REGION Network 79: K
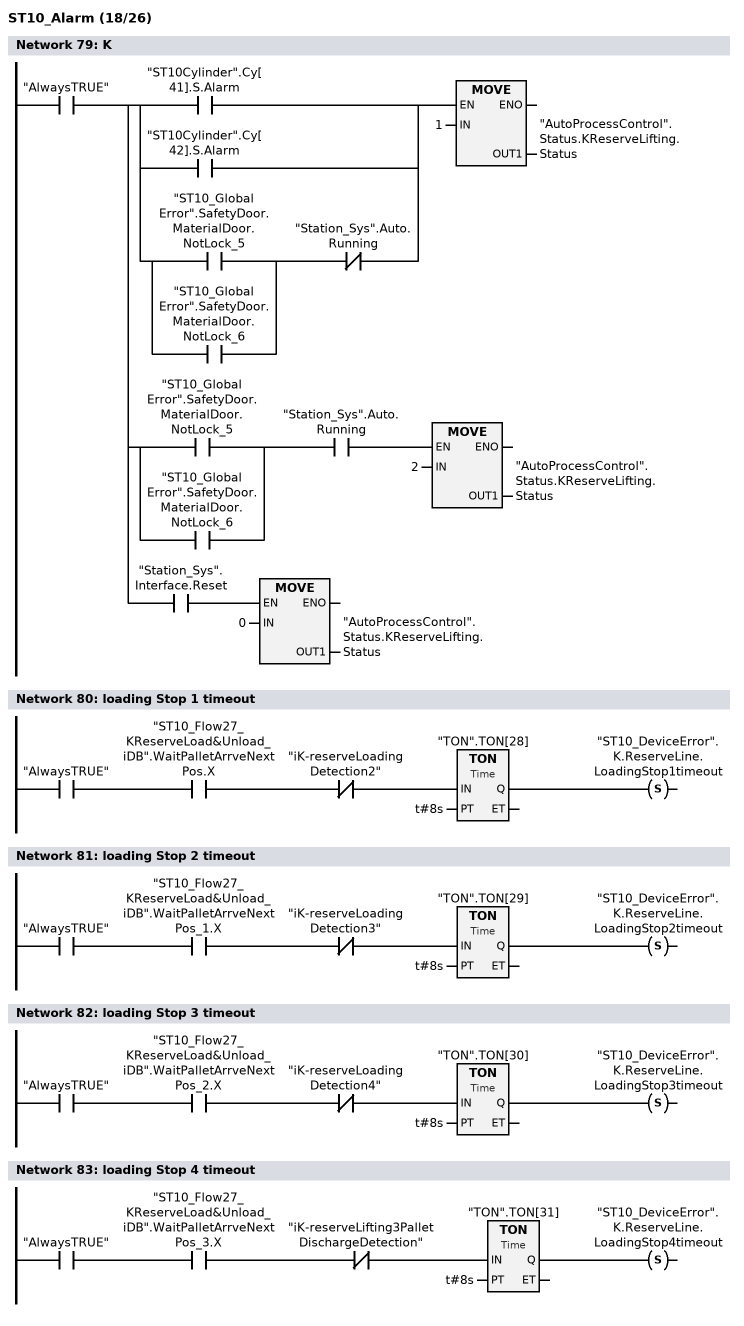
   RUNG wire#powerrail
      Contact( "AlwaysTRUE" )
      wire#w1
      Contact( "ST10Cylinder".Cy[41].S.Alarm )
      wire#w2
      Move(in := 1, out1 => "AutoProcessControl".Status.KReserveLifting.Status)
   END_RUNG
   RUNG wire#w1
      Contact( "ST10Cylinder".Cy[42].S.Alarm )
   END_RUNG wire#w2
   RUNG wire#w1
      Contact( "ST10_GlobalError".SafetyDoor.MaterialDoor.NotLock_5 )
      wire#w3
      I_Contact( "Station_Sys".Auto.Running )
   END_RUNG wire#w2
   RUNG wire#w1
      Contact( "ST10_GlobalError".SafetyDoor.MaterialDoor.NotLock_6 )
   END_RUNG wire#w3
   RUNG wire#w1
      Contact( "ST10_GlobalError".SafetyDoor.MaterialDoor.NotLock_5 )
      wire#w4
      Contact( "Station_Sys".Auto.Running )
      Move(in := 2, out1 => "AutoProcessControl".Status.KReserveLifting.Status)
   END_RUNG
   RUNG wire#w1
      Contact( "ST10_GlobalError".SafetyDoor.MaterialDoor.NotLock_6 )
   END_RUNG wire#w4
   RUNG wire#w1
      Contact( "Station_Sys".Interface.Reset )
      Move(in := 0, out1 => "AutoProcessControl".Status.KReserveLifting.Status)
   END_RUNG
   // the same network as SCL:
   IF "AlwaysTRUE" AND ("ST10Cylinder".Cy[41].S.Alarm OR "ST10Cylinder".Cy[42].S.Alarm OR (("ST10_GlobalError".SafetyDoor.MaterialDoor.NotLock_5 OR "ST10_GlobalError".SafetyDoor.MaterialDoor.NotLock_6) AND NOT "Station_Sys".Auto.Running)) THEN
       "AutoProcessControl".Status.KReserveLifting.Status := 1;
   END_IF;
   IF "AlwaysTRUE" AND ("ST10_GlobalError".SafetyDoor.MaterialDoor.NotLock_5 OR "ST10_GlobalError".SafetyDoor.MaterialDoor.NotLock_6) AND "Station_Sys".Auto.Running THEN
       "AutoProcessControl".Status.KReserveLifting.Status := 2;
   END_IF;
   IF "AlwaysTRUE" AND "Station_Sys".Interface.Reset THEN
       "AutoProcessControl".Status.KReserveLifting.Status := 0;
   END_IF;
END_REGION

REGION Network 80: loading Stop 1 timeout
   RUNG wire#powerrail
      Contact( "AlwaysTRUE" )
      Contact( "ST10_Flow27_KReserveLoad&Unload_iDB".WaitPalletArrveNextPos.X )
      I_Contact( "iK-reserveLoadingDetection2" )
      { S7_Templates := "time_type := Time" } "TON".TON[28].TON(pt := t#8s, et =>)
      S_Coil( "ST10_DeviceError".K.ReserveLine.LoadingStop1timeout )
   END_RUNG
   // the same network as SCL:
   "TON".TON[28].TON(IN := "AlwaysTRUE" AND "ST10_Flow27_KReserveLoad&Unload_iDB".WaitPalletArrveNextPos.X AND NOT "iK-reserveLoadingDetection2",
                     PT := t#8s);
   IF "TON".TON[28].Q THEN "ST10_DeviceError".K.ReserveLine.LoadingStop1timeout := TRUE; END_IF;
END_REGION

REGION Network 81: loading Stop 2 timeout
   RUNG wire#powerrail
      Contact( "AlwaysTRUE" )
      Contact( "ST10_Flow27_KReserveLoad&Unload_iDB".WaitPalletArrveNextPos_1.X )
      I_Contact( "iK-reserveLoadingDetection3" )
      { S7_Templates := "time_type := Time" } "TON".TON[29].TON(pt := t#8s, et =>)
      S_Coil( "ST10_DeviceError".K.ReserveLine.LoadingStop2timeout )
   END_RUNG
   // the same network as SCL:
   "TON".TON[29].TON(IN := "AlwaysTRUE" AND "ST10_Flow27_KReserveLoad&Unload_iDB".WaitPalletArrveNextPos_1.X AND NOT "iK-reserveLoadingDetection3",
                     PT := t#8s);
   IF "TON".TON[29].Q THEN "ST10_DeviceError".K.ReserveLine.LoadingStop2timeout := TRUE; END_IF;
END_REGION

REGION Network 82: loading Stop 3 timeout
   RUNG wire#powerrail
      Contact( "AlwaysTRUE" )
      Contact( "ST10_Flow27_KReserveLoad&Unload_iDB".WaitPalletArrveNextPos_2.X )
      I_Contact( "iK-reserveLoadingDetection4" )
      { S7_Templates := "time_type := Time" } "TON".TON[30].TON(pt := t#8s, et =>)
      S_Coil( "ST10_DeviceError".K.ReserveLine.LoadingStop3timeout )
   END_RUNG
   // the same network as SCL:
   "TON".TON[30].TON(IN := "AlwaysTRUE" AND "ST10_Flow27_KReserveLoad&Unload_iDB".WaitPalletArrveNextPos_2.X AND NOT "iK-reserveLoadingDetection4",
                     PT := t#8s);
   IF "TON".TON[30].Q THEN "ST10_DeviceError".K.ReserveLine.LoadingStop3timeout := TRUE; END_IF;
END_REGION

REGION Network 83: loading Stop 4 timeout
   RUNG wire#powerrail
      Contact( "AlwaysTRUE" )
      Contact( "ST10_Flow27_KReserveLoad&Unload_iDB".WaitPalletArrveNextPos_3.X )
      I_Contact( "iK-reserveLifting3PalletDischargeDetection" )
      { S7_Templates := "time_type := Time" } "TON".TON[31].TON(pt := t#8s, et =>)
      S_Coil( "ST10_DeviceError".K.ReserveLine.LoadingStop4timeout )
   END_RUNG
   // the same network as SCL:
   "TON".TON[31].TON(IN := "AlwaysTRUE" AND "ST10_Flow27_KReserveLoad&Unload_iDB".WaitPalletArrveNextPos_3.X AND NOT "iK-reserveLifting3PalletDischargeDetection",
                     PT := t#8s);
   IF "TON".TON[31].Q THEN "ST10_DeviceError".K.ReserveLine.LoadingStop4timeout := TRUE; END_IF;
END_REGION

REGION Network 84: unLoading Stop1 timeout
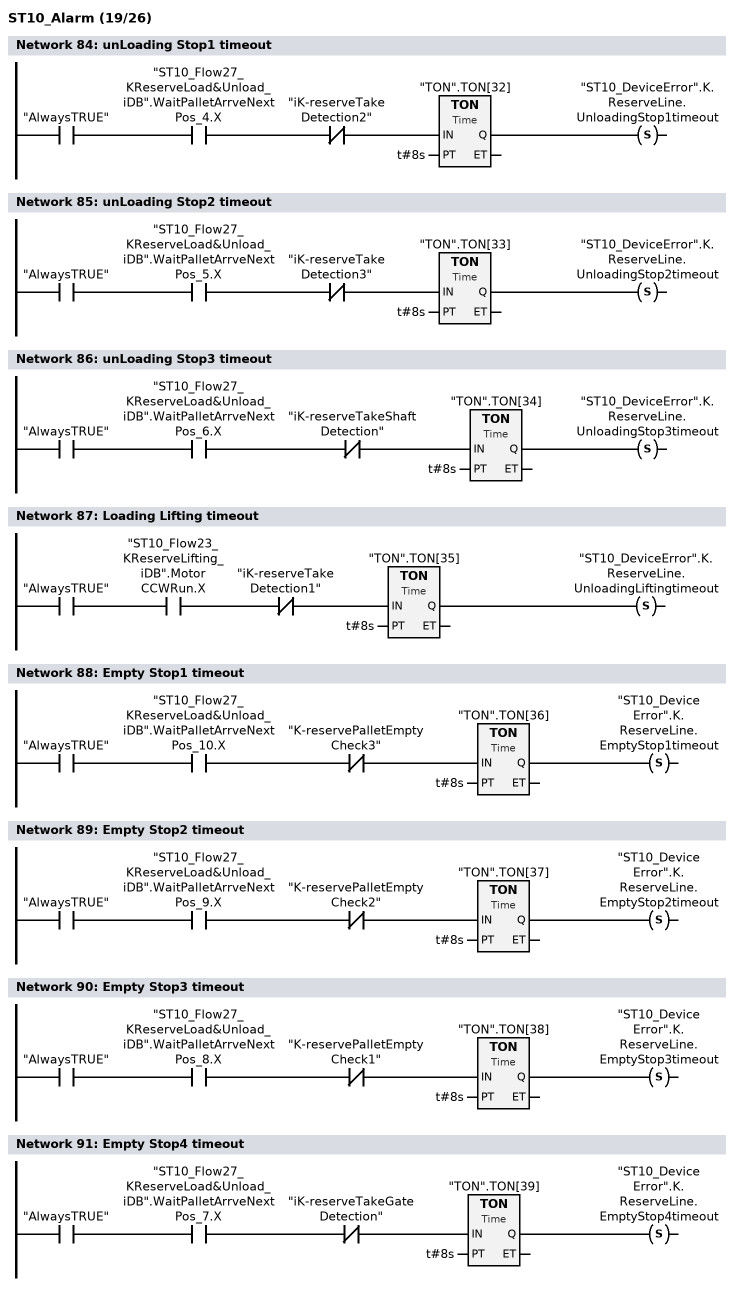
   RUNG wire#powerrail
      Contact( "AlwaysTRUE" )
      Contact( "ST10_Flow27_KReserveLoad&Unload_iDB".WaitPalletArrveNextPos_4.X )
      I_Contact( "iK-reserveTakeDetection2" )
      { S7_Templates := "time_type := Time" } "TON".TON[32].TON(pt := t#8s, et =>)
      S_Coil( "ST10_DeviceError".K.ReserveLine.UnloadingStop1timeout )
   END_RUNG
   // the same network as SCL:
   "TON".TON[32].TON(IN := "AlwaysTRUE" AND "ST10_Flow27_KReserveLoad&Unload_iDB".WaitPalletArrveNextPos_4.X AND NOT "iK-reserveTakeDetection2",
                     PT := t#8s);
   IF "TON".TON[32].Q THEN "ST10_DeviceError".K.ReserveLine.UnloadingStop1timeout := TRUE; END_IF;
END_REGION

REGION Network 85: unLoading Stop2 timeout
   RUNG wire#powerrail
      Contact( "AlwaysTRUE" )
      Contact( "ST10_Flow27_KReserveLoad&Unload_iDB".WaitPalletArrveNextPos_5.X )
      I_Contact( "iK-reserveTakeDetection3" )
      { S7_Templates := "time_type := Time" } "TON".TON[33].TON(pt := t#8s, et =>)
      S_Coil( "ST10_DeviceError".K.ReserveLine.UnloadingStop2timeout )
   END_RUNG
   // the same network as SCL:
   "TON".TON[33].TON(IN := "AlwaysTRUE" AND "ST10_Flow27_KReserveLoad&Unload_iDB".WaitPalletArrveNextPos_5.X AND NOT "iK-reserveTakeDetection3",
                     PT := t#8s);
   IF "TON".TON[33].Q THEN "ST10_DeviceError".K.ReserveLine.UnloadingStop2timeout := TRUE; END_IF;
END_REGION

REGION Network 86: unLoading Stop3 timeout
   RUNG wire#powerrail
      Contact( "AlwaysTRUE" )
      Contact( "ST10_Flow27_KReserveLoad&Unload_iDB".WaitPalletArrveNextPos_6.X )
      I_Contact( "iK-reserveTakeShaftDetection" )
      { S7_Templates := "time_type := Time" } "TON".TON[34].TON(pt := t#8s, et =>)
      S_Coil( "ST10_DeviceError".K.ReserveLine.UnloadingStop3timeout )
   END_RUNG
   // the same network as SCL:
   "TON".TON[34].TON(IN := "AlwaysTRUE" AND "ST10_Flow27_KReserveLoad&Unload_iDB".WaitPalletArrveNextPos_6.X AND NOT "iK-reserveTakeShaftDetection",
                     PT := t#8s);
   IF "TON".TON[34].Q THEN "ST10_DeviceError".K.ReserveLine.UnloadingStop3timeout := TRUE; END_IF;
END_REGION

REGION Network 87: Loading Lifting timeout
   RUNG wire#powerrail
      Contact( "AlwaysTRUE" )
      Contact( "ST10_Flow23_KReserveLifting_iDB".MotorCCWRun.X )
      I_Contact( "iK-reserveTakeDetection1" )
      { S7_Templates := "time_type := Time" } "TON".TON[35].TON(pt := t#8s, et =>)
      S_Coil( "ST10_DeviceError".K.ReserveLine.UnloadingLiftingtimeout )
   END_RUNG
   // the same network as SCL:
   "TON".TON[35].TON(IN := "AlwaysTRUE" AND "ST10_Flow23_KReserveLifting_iDB".MotorCCWRun.X AND NOT "iK-reserveTakeDetection1",
                     PT := t#8s);
   IF "TON".TON[35].Q THEN "ST10_DeviceError".K.ReserveLine.UnloadingLiftingtimeout := TRUE; END_IF;
END_REGION

REGION Network 88: Empty Stop1 timeout
   RUNG wire#powerrail
      Contact( "AlwaysTRUE" )
      Contact( "ST10_Flow27_KReserveLoad&Unload_iDB".WaitPalletArrveNextPos_10.X )
      I_Contact( "K-reservePalletEmptyCheck3" )
      { S7_Templates := "time_type := Time" } "TON".TON[36].TON(pt := t#8s, et =>)
      S_Coil( "ST10_DeviceError".K.ReserveLine.EmptyStop1timeout )
   END_RUNG
   // the same network as SCL:
   "TON".TON[36].TON(IN := "AlwaysTRUE" AND "ST10_Flow27_KReserveLoad&Unload_iDB".WaitPalletArrveNextPos_10.X AND NOT "K-reservePalletEmptyCheck3",
                     PT := t#8s);
   IF "TON".TON[36].Q THEN "ST10_DeviceError".K.ReserveLine.EmptyStop1timeout := TRUE; END_IF;
END_REGION

REGION Network 89: Empty Stop2 timeout
   RUNG wire#powerrail
      Contact( "AlwaysTRUE" )
      Contact( "ST10_Flow27_KReserveLoad&Unload_iDB".WaitPalletArrveNextPos_9.X )
      I_Contact( "K-reservePalletEmptyCheck2" )
      { S7_Templates := "time_type := Time" } "TON".TON[37].TON(pt := t#8s, et =>)
      S_Coil( "ST10_DeviceError".K.ReserveLine.EmptyStop2timeout )
   END_RUNG
   // the same network as SCL:
   "TON".TON[37].TON(IN := "AlwaysTRUE" AND "ST10_Flow27_KReserveLoad&Unload_iDB".WaitPalletArrveNextPos_9.X AND NOT "K-reservePalletEmptyCheck2",
                     PT := t#8s);
   IF "TON".TON[37].Q THEN "ST10_DeviceError".K.ReserveLine.EmptyStop2timeout := TRUE; END_IF;
END_REGION

REGION Network 90: Empty Stop3 timeout
   RUNG wire#powerrail
      Contact( "AlwaysTRUE" )
      Contact( "ST10_Flow27_KReserveLoad&Unload_iDB".WaitPalletArrveNextPos_8.X )
      I_Contact( "K-reservePalletEmptyCheck1" )
      { S7_Templates := "time_type := Time" } "TON".TON[38].TON(pt := t#8s, et =>)
      S_Coil( "ST10_DeviceError".K.ReserveLine.EmptyStop3timeout )
   END_RUNG
   // the same network as SCL:
   "TON".TON[38].TON(IN := "AlwaysTRUE" AND "ST10_Flow27_KReserveLoad&Unload_iDB".WaitPalletArrveNextPos_8.X AND NOT "K-reservePalletEmptyCheck1",
                     PT := t#8s);
   IF "TON".TON[38].Q THEN "ST10_DeviceError".K.ReserveLine.EmptyStop3timeout := TRUE; END_IF;
END_REGION

REGION Network 91: Empty Stop4 timeout
   RUNG wire#powerrail
      Contact( "AlwaysTRUE" )
      Contact( "ST10_Flow27_KReserveLoad&Unload_iDB".WaitPalletArrveNextPos_7.X )
      I_Contact( "iK-reserveTakeGateDetection" )
      { S7_Templates := "time_type := Time" } "TON".TON[39].TON(pt := t#8s, et =>)
      S_Coil( "ST10_DeviceError".K.ReserveLine.EmptyStop4timeout )
   END_RUNG
   // the same network as SCL:
   "TON".TON[39].TON(IN := "AlwaysTRUE" AND "ST10_Flow27_KReserveLoad&Unload_iDB".WaitPalletArrveNextPos_7.X AND NOT "iK-reserveTakeGateDetection",
                     PT := t#8s);
   IF "TON".TON[39].Q THEN "ST10_DeviceError".K.ReserveLine.EmptyStop4timeout := TRUE; END_IF;
END_REGION

REGION Network 93: ******************** L_Unloading ********************
END_REGION

REGION Network 94: L
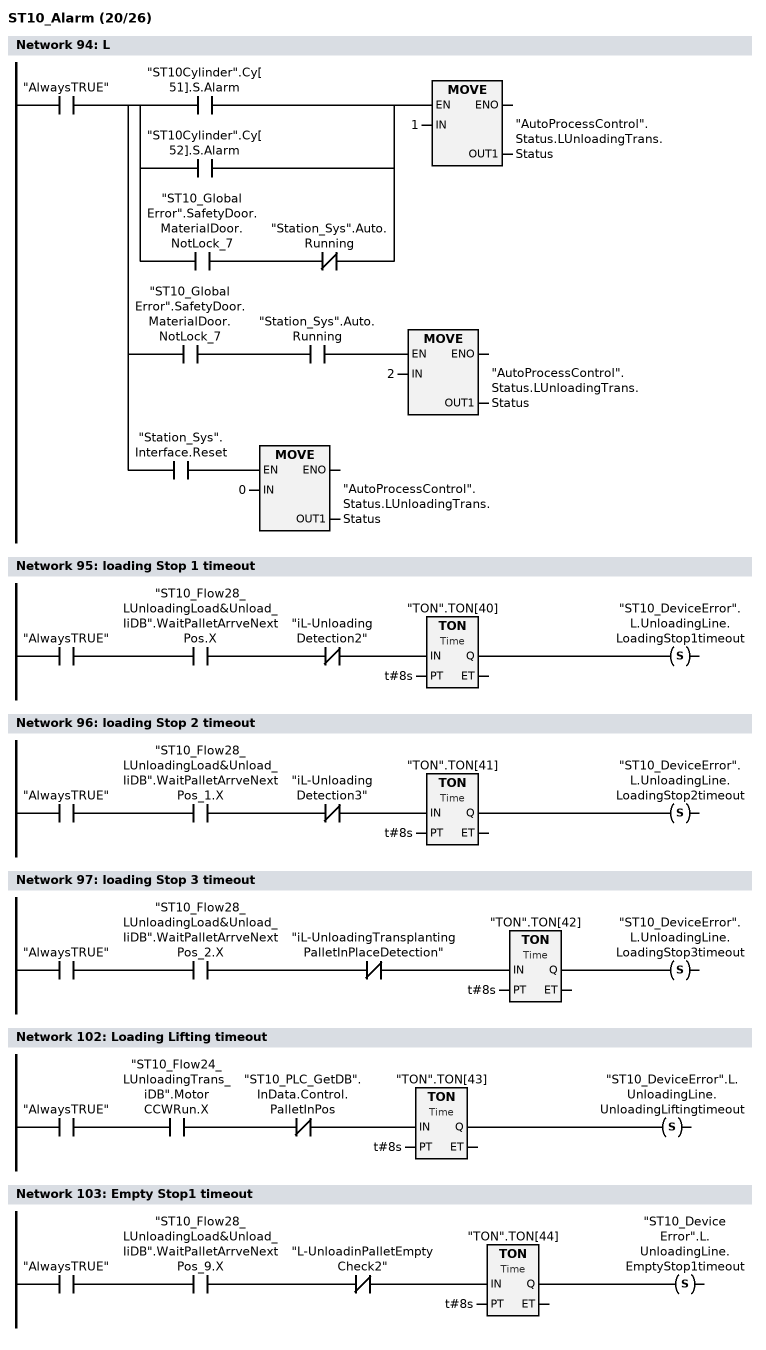
   RUNG wire#powerrail
      Contact( "AlwaysTRUE" )
      wire#w1
      Contact( "ST10Cylinder".Cy[51].S.Alarm )
      wire#w2
      Move(in := 1, out1 => "AutoProcessControl".Status.LUnloadingTrans.Status)
   END_RUNG
   RUNG wire#w1
      Contact( "ST10Cylinder".Cy[52].S.Alarm )
   END_RUNG wire#w2
   RUNG wire#w1
      Contact( "ST10_GlobalError".SafetyDoor.MaterialDoor.NotLock_7 )
      I_Contact( "Station_Sys".Auto.Running )
   END_RUNG wire#w2
   RUNG wire#w1
      Contact( "ST10_GlobalError".SafetyDoor.MaterialDoor.NotLock_7 )
      Contact( "Station_Sys".Auto.Running )
      Move(in := 2, out1 => "AutoProcessControl".Status.LUnloadingTrans.Status)
   END_RUNG
   RUNG wire#w1
      Contact( "Station_Sys".Interface.Reset )
      Move(in := 0, out1 => "AutoProcessControl".Status.LUnloadingTrans.Status)
   END_RUNG
   // the same network as SCL:
   IF "AlwaysTRUE" AND ("ST10Cylinder".Cy[51].S.Alarm OR "ST10Cylinder".Cy[52].S.Alarm OR ("ST10_GlobalError".SafetyDoor.MaterialDoor.NotLock_7 AND NOT "Station_Sys".Auto.Running)) THEN
       "AutoProcessControl".Status.LUnloadingTrans.Status := 1;
   END_IF;
   IF "AlwaysTRUE" AND "ST10_GlobalError".SafetyDoor.MaterialDoor.NotLock_7 AND "Station_Sys".Auto.Running THEN
       "AutoProcessControl".Status.LUnloadingTrans.Status := 2;
   END_IF;
   IF "AlwaysTRUE" AND "Station_Sys".Interface.Reset THEN
       "AutoProcessControl".Status.LUnloadingTrans.Status := 0;
   END_IF;
END_REGION

REGION Network 95: loading Stop 1 timeout
   RUNG wire#powerrail
      Contact( "AlwaysTRUE" )
      Contact( "ST10_Flow28_LUnloadingLoad&Unload_IiDB".WaitPalletArrveNextPos.X )
      I_Contact( "iL-UnloadingDetection2" )
      { S7_Templates := "time_type := Time" } "TON".TON[40].TON(pt := t#8s, et =>)
      S_Coil( "ST10_DeviceError".L.UnloadingLine.LoadingStop1timeout )
   END_RUNG
   // the same network as SCL:
   "TON".TON[40].TON(IN := "AlwaysTRUE" AND "ST10_Flow28_LUnloadingLoad&Unload_IiDB".WaitPalletArrveNextPos.X AND NOT "iL-UnloadingDetection2",
                     PT := t#8s);
   IF "TON".TON[40].Q THEN "ST10_DeviceError".L.UnloadingLine.LoadingStop1timeout := TRUE; END_IF;
END_REGION

REGION Network 96: loading Stop 2 timeout
   RUNG wire#powerrail
      Contact( "AlwaysTRUE" )
      Contact( "ST10_Flow28_LUnloadingLoad&Unload_IiDB".WaitPalletArrveNextPos_1.X )
      I_Contact( "iL-UnloadingDetection3" )
      { S7_Templates := "time_type := Time" } "TON".TON[41].TON(pt := t#8s, et =>)
      S_Coil( "ST10_DeviceError".L.UnloadingLine.LoadingStop2timeout )
   END_RUNG
   // the same network as SCL:
   "TON".TON[41].TON(IN := "AlwaysTRUE" AND "ST10_Flow28_LUnloadingLoad&Unload_IiDB".WaitPalletArrveNextPos_1.X AND NOT "iL-UnloadingDetection3",
                     PT := t#8s);
   IF "TON".TON[41].Q THEN "ST10_DeviceError".L.UnloadingLine.LoadingStop2timeout := TRUE; END_IF;
END_REGION

REGION Network 97: loading Stop 3 timeout
   RUNG wire#powerrail
      Contact( "AlwaysTRUE" )
      Contact( "ST10_Flow28_LUnloadingLoad&Unload_IiDB".WaitPalletArrveNextPos_2.X )
      I_Contact( "iL-UnloadingTransplantingPalletInPlaceDetection" )
      { S7_Templates := "time_type := Time" } "TON".TON[42].TON(pt := t#8s, et =>)
      S_Coil( "ST10_DeviceError".L.UnloadingLine.LoadingStop3timeout )
   END_RUNG
   // the same network as SCL:
   "TON".TON[42].TON(IN := "AlwaysTRUE" AND "ST10_Flow28_LUnloadingLoad&Unload_IiDB".WaitPalletArrveNextPos_2.X AND NOT "iL-UnloadingTransplantingPalletInPlaceDetection",
                     PT := t#8s);
   IF "TON".TON[42].Q THEN "ST10_DeviceError".L.UnloadingLine.LoadingStop3timeout := TRUE; END_IF;
END_REGION

REGION Network 98: loading Stop 4 timeout
END_REGION

REGION Network 99: unLoading Stop1 timeout
END_REGION

REGION Network 100: unLoading Stop2 timeout
END_REGION

REGION Network 101: unLoading Stop3 timeout
END_REGION

REGION Network 102: Loading Lifting timeout
   RUNG wire#powerrail
      Contact( "AlwaysTRUE" )
      Contact( "ST10_Flow24_LUnloadingTrans_iDB".MotorCCWRun.X )
      I_Contact( "ST10_PLC_GetDB".InData.Control.PalletInPos )
      { S7_Templates := "time_type := Time" } "TON".TON[43].TON(pt := t#8s, et =>)
      S_Coil( "ST10_DeviceError".L.UnloadingLine.UnloadingLiftingtimeout )
   END_RUNG
   // the same network as SCL:
   "TON".TON[43].TON(IN := "AlwaysTRUE" AND "ST10_Flow24_LUnloadingTrans_iDB".MotorCCWRun.X AND NOT "ST10_PLC_GetDB".InData.Control.PalletInPos,
                     PT := t#8s);
   IF "TON".TON[43].Q THEN "ST10_DeviceError".L.UnloadingLine.UnloadingLiftingtimeout := TRUE; END_IF;
END_REGION

REGION Network 103: Empty Stop1 timeout
   RUNG wire#powerrail
      Contact( "AlwaysTRUE" )
      Contact( "ST10_Flow28_LUnloadingLoad&Unload_IiDB".WaitPalletArrveNextPos_9.X )
      I_Contact( "L-UnloadinPalletEmptyCheck2" )
      { S7_Templates := "time_type := Time" } "TON".TON[44].TON(pt := t#8s, et =>)
      S_Coil( "ST10_DeviceError".L.UnloadingLine.EmptyStop1timeout )
   END_RUNG
   // the same network as SCL:
   "TON".TON[44].TON(IN := "AlwaysTRUE" AND "ST10_Flow28_LUnloadingLoad&Unload_IiDB".WaitPalletArrveNextPos_9.X AND NOT "L-UnloadinPalletEmptyCheck2",
                     PT := t#8s);
   IF "TON".TON[44].Q THEN "ST10_DeviceError".L.UnloadingLine.EmptyStop1timeout := TRUE; END_IF;
END_REGION

REGION Network 104: Empty Stop2 timeout
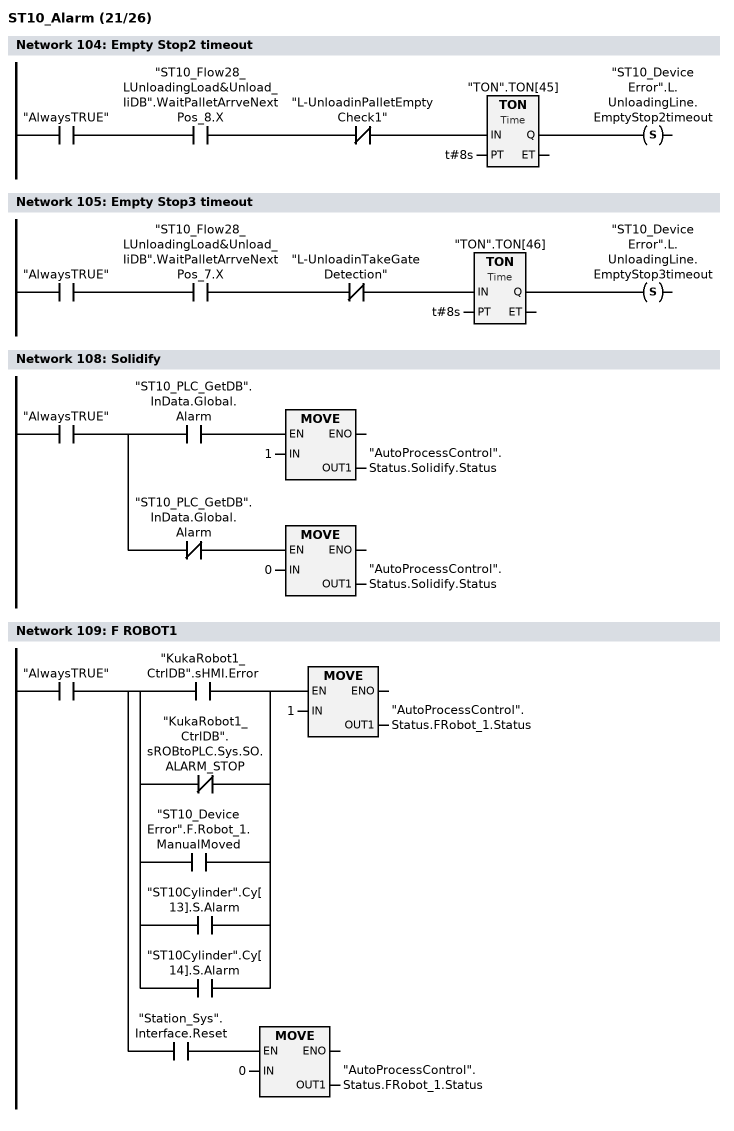
   RUNG wire#powerrail
      Contact( "AlwaysTRUE" )
      Contact( "ST10_Flow28_LUnloadingLoad&Unload_IiDB".WaitPalletArrveNextPos_8.X )
      I_Contact( "L-UnloadinPalletEmptyCheck1" )
      { S7_Templates := "time_type := Time" } "TON".TON[45].TON(pt := t#8s, et =>)
      S_Coil( "ST10_DeviceError".L.UnloadingLine.EmptyStop2timeout )
   END_RUNG
   // the same network as SCL:
   "TON".TON[45].TON(IN := "AlwaysTRUE" AND "ST10_Flow28_LUnloadingLoad&Unload_IiDB".WaitPalletArrveNextPos_8.X AND NOT "L-UnloadinPalletEmptyCheck1",
                     PT := t#8s);
   IF "TON".TON[45].Q THEN "ST10_DeviceError".L.UnloadingLine.EmptyStop2timeout := TRUE; END_IF;
END_REGION

REGION Network 105: Empty Stop3 timeout
   RUNG wire#powerrail
      Contact( "AlwaysTRUE" )
      Contact( "ST10_Flow28_LUnloadingLoad&Unload_IiDB".WaitPalletArrveNextPos_7.X )
      I_Contact( "L-UnloadinTakeGateDetection" )
      { S7_Templates := "time_type := Time" } "TON".TON[46].TON(pt := t#8s, et =>)
      S_Coil( "ST10_DeviceError".L.UnloadingLine.EmptyStop3timeout )
   END_RUNG
   // the same network as SCL:
   "TON".TON[46].TON(IN := "AlwaysTRUE" AND "ST10_Flow28_LUnloadingLoad&Unload_IiDB".WaitPalletArrveNextPos_7.X AND NOT "L-UnloadinTakeGateDetection",
                     PT := t#8s);
   IF "TON".TON[46].Q THEN "ST10_DeviceError".L.UnloadingLine.EmptyStop3timeout := TRUE; END_IF;
END_REGION

REGION Network 106: Empty Stop4 timeout
END_REGION

REGION Network 108: Solidify
   RUNG wire#powerrail
      Contact( "AlwaysTRUE" )
      wire#w1
      Contact( "ST10_PLC_GetDB".InData.Global.Alarm )
      Move(in := 1, out1 => "AutoProcessControl".Status.Solidify.Status)
   END_RUNG
   RUNG wire#w1
      I_Contact( "ST10_PLC_GetDB".InData.Global.Alarm )
      Move(in := 0, out1 => "AutoProcessControl".Status.Solidify.Status)
   END_RUNG
   // the same network as SCL:
   IF "AlwaysTRUE" AND "ST10_PLC_GetDB".InData.Global.Alarm THEN
       "AutoProcessControl".Status.Solidify.Status := 1;
   END_IF;
   IF "AlwaysTRUE" AND NOT "ST10_PLC_GetDB".InData.Global.Alarm THEN
       "AutoProcessControl".Status.Solidify.Status := 0;
   END_IF;
END_REGION

REGION Network 109: F ROBOT1
   RUNG wire#powerrail
      Contact( "AlwaysTRUE" )
      wire#w1
      Contact( "KukaRobot1_CtrlDB".sHMI.Error )
      wire#w2
      Move(in := 1, out1 => "AutoProcessControl".Status.FRobot_1.Status)
   END_RUNG
   RUNG wire#w1
      I_Contact( "KukaRobot1_CtrlDB".sROBtoPLC.Sys.SO.ALARM_STOP )
   END_RUNG wire#w2
   RUNG wire#w1
      Contact( "ST10_DeviceError".F.Robot_1.ManualMoved )
   END_RUNG wire#w2
   RUNG wire#w1
      Contact( "ST10Cylinder".Cy[13].S.Alarm )
   END_RUNG wire#w2
   RUNG wire#w1
      Contact( "ST10Cylinder".Cy[14].S.Alarm )
   END_RUNG wire#w2
   RUNG wire#w1
      Contact( "Station_Sys".Interface.Reset )
      Move(in := 0, out1 => "AutoProcessControl".Status.FRobot_1.Status)
   END_RUNG
   // the same network as SCL:
   IF "AlwaysTRUE" AND ("KukaRobot1_CtrlDB".sHMI.Error OR NOT "KukaRobot1_CtrlDB".sROBtoPLC.Sys.SO.ALARM_STOP OR "ST10_DeviceError".F.Robot_1.ManualMoved OR "ST10Cylinder".Cy[13].S.Alarm OR "ST10Cylinder".Cy[14].S.Alarm) THEN
       "AutoProcessControl".Status.FRobot_1.Status := 1;
   END_IF;
   IF "AlwaysTRUE" AND "Station_Sys".Interface.Reset THEN
       "AutoProcessControl".Status.FRobot_1.Status := 0;
   END_IF;
END_REGION

REGION Network 110: F ROBOT2
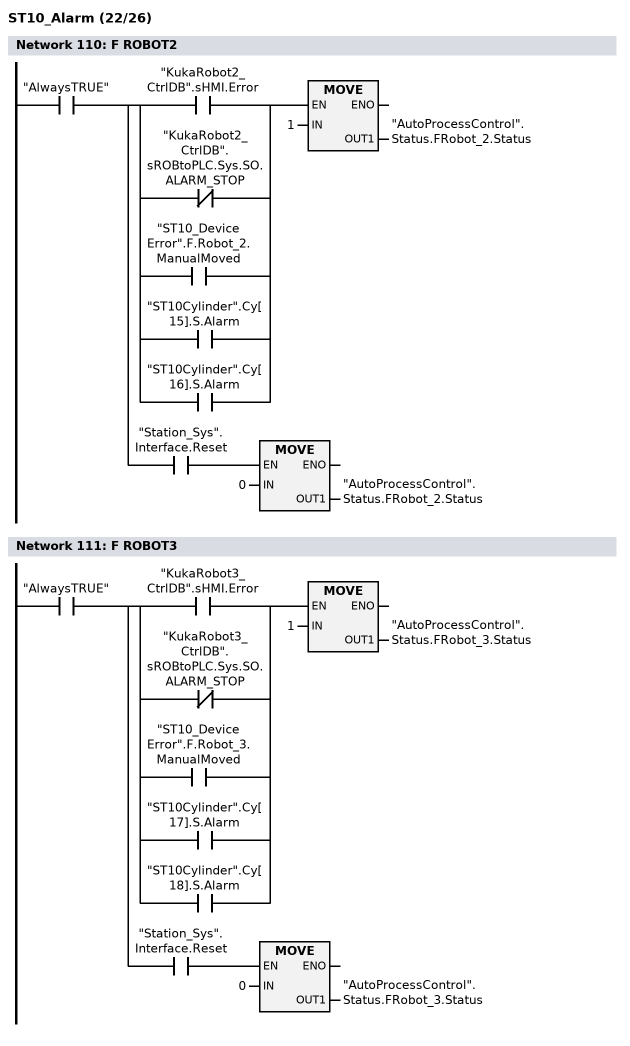
   RUNG wire#powerrail
      Contact( "AlwaysTRUE" )
      wire#w1
      Contact( "KukaRobot2_CtrlDB".sHMI.Error )
      wire#w2
      Move(in := 1, out1 => "AutoProcessControl".Status.FRobot_2.Status)
   END_RUNG
   RUNG wire#w1
      I_Contact( "KukaRobot2_CtrlDB".sROBtoPLC.Sys.SO.ALARM_STOP )
   END_RUNG wire#w2
   RUNG wire#w1
      Contact( "ST10_DeviceError".F.Robot_2.ManualMoved )
   END_RUNG wire#w2
   RUNG wire#w1
      Contact( "ST10Cylinder".Cy[15].S.Alarm )
   END_RUNG wire#w2
   RUNG wire#w1
      Contact( "ST10Cylinder".Cy[16].S.Alarm )
   END_RUNG wire#w2
   RUNG wire#w1
      Contact( "Station_Sys".Interface.Reset )
      Move(in := 0, out1 => "AutoProcessControl".Status.FRobot_2.Status)
   END_RUNG
   // the same network as SCL:
   IF "AlwaysTRUE" AND ("KukaRobot2_CtrlDB".sHMI.Error OR NOT "KukaRobot2_CtrlDB".sROBtoPLC.Sys.SO.ALARM_STOP OR "ST10_DeviceError".F.Robot_2.ManualMoved OR "ST10Cylinder".Cy[15].S.Alarm OR "ST10Cylinder".Cy[16].S.Alarm) THEN
       "AutoProcessControl".Status.FRobot_2.Status := 1;
   END_IF;
   IF "AlwaysTRUE" AND "Station_Sys".Interface.Reset THEN
       "AutoProcessControl".Status.FRobot_2.Status := 0;
   END_IF;
END_REGION

REGION Network 111: F ROBOT3
   RUNG wire#powerrail
      Contact( "AlwaysTRUE" )
      wire#w1
      Contact( "KukaRobot3_CtrlDB".sHMI.Error )
      wire#w2
      Move(in := 1, out1 => "AutoProcessControl".Status.FRobot_3.Status)
   END_RUNG
   RUNG wire#w1
      I_Contact( "KukaRobot3_CtrlDB".sROBtoPLC.Sys.SO.ALARM_STOP )
   END_RUNG wire#w2
   RUNG wire#w1
      Contact( "ST10_DeviceError".F.Robot_3.ManualMoved )
   END_RUNG wire#w2
   RUNG wire#w1
      Contact( "ST10Cylinder".Cy[17].S.Alarm )
   END_RUNG wire#w2
   RUNG wire#w1
      Contact( "ST10Cylinder".Cy[18].S.Alarm )
   END_RUNG wire#w2
   RUNG wire#w1
      Contact( "Station_Sys".Interface.Reset )
      Move(in := 0, out1 => "AutoProcessControl".Status.FRobot_3.Status)
   END_RUNG
   // the same network as SCL:
   IF "AlwaysTRUE" AND ("KukaRobot3_CtrlDB".sHMI.Error OR NOT "KukaRobot3_CtrlDB".sROBtoPLC.Sys.SO.ALARM_STOP OR "ST10_DeviceError".F.Robot_3.ManualMoved OR "ST10Cylinder".Cy[17].S.Alarm OR "ST10Cylinder".Cy[18].S.Alarm) THEN
       "AutoProcessControl".Status.FRobot_3.Status := 1;
   END_IF;
   IF "AlwaysTRUE" AND "Station_Sys".Interface.Reset THEN
       "AutoProcessControl".Status.FRobot_3.Status := 0;
   END_IF;
END_REGION

REGION Network 112: ******************** E NG ********************
END_REGION

REGION Network 113: E NG_1
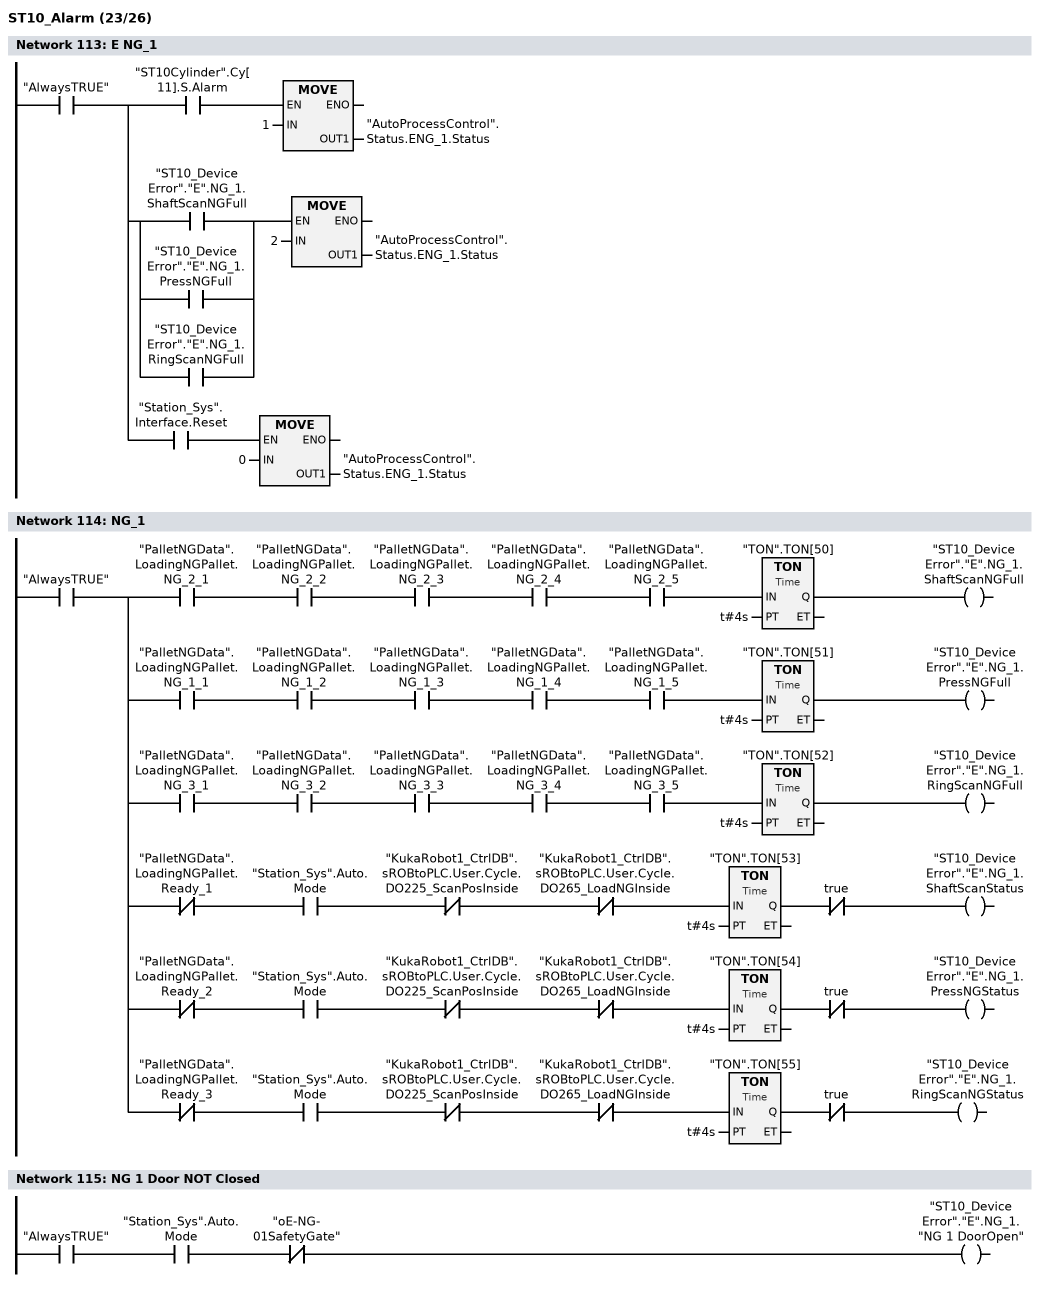
   RUNG wire#powerrail
      Contact( "AlwaysTRUE" )
      wire#w1
      Contact( "ST10Cylinder".Cy[11].S.Alarm )
      Move(in := 1, out1 => "AutoProcessControl".Status.ENG_1.Status)
   END_RUNG
   RUNG wire#w1
      Contact( "ST10_DeviceError"."E".NG_1.ShaftScanNGFull )
      wire#w2
      Move(in := 2, out1 => "AutoProcessControl".Status.ENG_1.Status)
   END_RUNG
   RUNG wire#w1
      Contact( "ST10_DeviceError"."E".NG_1.PressNGFull )
   END_RUNG wire#w2
   RUNG wire#w1
      Contact( "ST10_DeviceError"."E".NG_1.RingScanNGFull )
   END_RUNG wire#w2
   RUNG wire#w1
      Contact( "Station_Sys".Interface.Reset )
      Move(in := 0, out1 => "AutoProcessControl".Status.ENG_1.Status)
   END_RUNG
   // the same network as SCL:
   IF "AlwaysTRUE" AND "ST10Cylinder".Cy[11].S.Alarm THEN
       "AutoProcessControl".Status.ENG_1.Status := 1;
   END_IF;
   IF "AlwaysTRUE" AND ("ST10_DeviceError"."E".NG_1.ShaftScanNGFull OR "ST10_DeviceError"."E".NG_1.PressNGFull OR "ST10_DeviceError"."E".NG_1.RingScanNGFull) THEN
       "AutoProcessControl".Status.ENG_1.Status := 2;
   END_IF;
   IF "AlwaysTRUE" AND "Station_Sys".Interface.Reset THEN
       "AutoProcessControl".Status.ENG_1.Status := 0;
   END_IF;
END_REGION

REGION Network 114: NG_1
   RUNG wire#powerrail
      Contact( "AlwaysTRUE" )
      wire#w1
      Contact( "PalletNGData".LoadingNGPallet.NG_2_1 )
      Contact( "PalletNGData".LoadingNGPallet.NG_2_2 )
      Contact( "PalletNGData".LoadingNGPallet.NG_2_3 )
      Contact( "PalletNGData".LoadingNGPallet.NG_2_4 )
      Contact( "PalletNGData".LoadingNGPallet.NG_2_5 )
      { S7_Templates := "time_type := Time" } "TON".TON[50].TON(pt := t#4s, et =>)
      Coil( "ST10_DeviceError"."E".NG_1.ShaftScanNGFull )
   END_RUNG
   RUNG wire#w1
      Contact( "PalletNGData".LoadingNGPallet.NG_1_1 )
      Contact( "PalletNGData".LoadingNGPallet.NG_1_2 )
      Contact( "PalletNGData".LoadingNGPallet.NG_1_3 )
      Contact( "PalletNGData".LoadingNGPallet.NG_1_4 )
      Contact( "PalletNGData".LoadingNGPallet.NG_1_5 )
      { S7_Templates := "time_type := Time" } "TON".TON[51].TON(pt := t#4s, et =>)
      Coil( "ST10_DeviceError"."E".NG_1.PressNGFull )
   END_RUNG
   RUNG wire#w1
      Contact( "PalletNGData".LoadingNGPallet.NG_3_1 )
      Contact( "PalletNGData".LoadingNGPallet.NG_3_2 )
      Contact( "PalletNGData".LoadingNGPallet.NG_3_3 )
      Contact( "PalletNGData".LoadingNGPallet.NG_3_4 )
      Contact( "PalletNGData".LoadingNGPallet.NG_3_5 )
      { S7_Templates := "time_type := Time" } "TON".TON[52].TON(pt := t#4s, et =>)
      Coil( "ST10_DeviceError"."E".NG_1.RingScanNGFull )
   END_RUNG
   RUNG wire#w1
      I_Contact( "PalletNGData".LoadingNGPallet.Ready_1 )
      Contact( "Station_Sys".Auto.Mode )
      I_Contact( "KukaRobot1_CtrlDB".sROBtoPLC.User.Cycle.DO225_ScanPosInside )
      I_Contact( "KukaRobot1_CtrlDB".sROBtoPLC.User.Cycle.DO265_LoadNGInside )
      { S7_Templates := "time_type := Time" } "TON".TON[53].TON(pt := t#4s, et =>)
      I_Contact( true )
      Coil( "ST10_DeviceError"."E".NG_1.ShaftScanStatus )
   END_RUNG
   RUNG wire#w1
      I_Contact( "PalletNGData".LoadingNGPallet.Ready_2 )
      Contact( "Station_Sys".Auto.Mode )
      I_Contact( "KukaRobot1_CtrlDB".sROBtoPLC.User.Cycle.DO225_ScanPosInside )
      I_Contact( "KukaRobot1_CtrlDB".sROBtoPLC.User.Cycle.DO265_LoadNGInside )
      { S7_Templates := "time_type := Time" } "TON".TON[54].TON(pt := t#4s, et =>)
      I_Contact( true )
      Coil( "ST10_DeviceError"."E".NG_1.PressNGStatus )
   END_RUNG
   RUNG wire#w1
      I_Contact( "PalletNGData".LoadingNGPallet.Ready_3 )
      Contact( "Station_Sys".Auto.Mode )
      I_Contact( "KukaRobot1_CtrlDB".sROBtoPLC.User.Cycle.DO225_ScanPosInside )
      I_Contact( "KukaRobot1_CtrlDB".sROBtoPLC.User.Cycle.DO265_LoadNGInside )
      { S7_Templates := "time_type := Time" } "TON".TON[55].TON(pt := t#4s, et =>)
      I_Contact( true )
      Coil( "ST10_DeviceError"."E".NG_1.RingScanNGStatus )
   END_RUNG
   // the same network as SCL:
   "TON".TON[50].TON(IN := "AlwaysTRUE" AND "PalletNGData".LoadingNGPallet.NG_2_1 AND "PalletNGData".LoadingNGPallet.NG_2_2 AND "PalletNGData".LoadingNGPallet.NG_2_3 AND "PalletNGData".LoadingNGPallet.NG_2_4 AND "PalletNGData".LoadingNGPallet.NG_2_5,
                     PT := t#4s);
   "ST10_DeviceError"."E".NG_1.ShaftScanNGFull := "TON".TON[50].Q;
   "TON".TON[51].TON(IN := "AlwaysTRUE" AND "PalletNGData".LoadingNGPallet.NG_1_1 AND "PalletNGData".LoadingNGPallet.NG_1_2 AND "PalletNGData".LoadingNGPallet.NG_1_3 AND "PalletNGData".LoadingNGPallet.NG_1_4 AND "PalletNGData".LoadingNGPallet.NG_1_5,
                     PT := t#4s);
   "ST10_DeviceError"."E".NG_1.PressNGFull := "TON".TON[51].Q;
   "TON".TON[52].TON(IN := "AlwaysTRUE" AND "PalletNGData".LoadingNGPallet.NG_3_1 AND "PalletNGData".LoadingNGPallet.NG_3_2 AND "PalletNGData".LoadingNGPallet.NG_3_3 AND "PalletNGData".LoadingNGPallet.NG_3_4 AND "PalletNGData".LoadingNGPallet.NG_3_5,
                     PT := t#4s);
   "ST10_DeviceError"."E".NG_1.RingScanNGFull := "TON".TON[52].Q;
   "TON".TON[53].TON(IN := "AlwaysTRUE" AND NOT "PalletNGData".LoadingNGPallet.Ready_1 AND "Station_Sys".Auto.Mode AND NOT "KukaRobot1_CtrlDB".sROBtoPLC.User.Cycle.DO225_ScanPosInside AND NOT "KukaRobot1_CtrlDB".sROBtoPLC.User.Cycle.DO265_LoadNGInside,
                     PT := t#4s);
   "ST10_DeviceError"."E".NG_1.ShaftScanStatus := "TON".TON[53].Q AND NOT true;
   "TON".TON[54].TON(IN := "AlwaysTRUE" AND NOT "PalletNGData".LoadingNGPallet.Ready_2 AND "Station_Sys".Auto.Mode AND NOT "KukaRobot1_CtrlDB".sROBtoPLC.User.Cycle.DO225_ScanPosInside AND NOT "KukaRobot1_CtrlDB".sROBtoPLC.User.Cycle.DO265_LoadNGInside,
                     PT := t#4s);
   "ST10_DeviceError"."E".NG_1.PressNGStatus := "TON".TON[54].Q AND NOT true;
   "TON".TON[55].TON(IN := "AlwaysTRUE" AND NOT "PalletNGData".LoadingNGPallet.Ready_3 AND "Station_Sys".Auto.Mode AND NOT "KukaRobot1_CtrlDB".sROBtoPLC.User.Cycle.DO225_ScanPosInside AND NOT "KukaRobot1_CtrlDB".sROBtoPLC.User.Cycle.DO265_LoadNGInside,
                     PT := t#4s);
   "ST10_DeviceError"."E".NG_1.RingScanNGStatus := "TON".TON[55].Q AND NOT true;
END_REGION

REGION Network 115: NG 1 Door NOT Closed
   RUNG wire#powerrail
      Contact( "AlwaysTRUE" )
      Contact( "Station_Sys".Auto.Mode )
      I_Contact( "oE-NG-01SafetyGate" )
      Coil( "ST10_DeviceError"."E".NG_1."NG 1 DoorOpen" )
   END_RUNG
   // the same network as SCL:
   "ST10_DeviceError"."E".NG_1."NG 1 DoorOpen" := "AlwaysTRUE" AND "Station_Sys".Auto.Mode AND NOT "oE-NG-01SafetyGate";
END_REGION

REGION Network 116: E NG_2
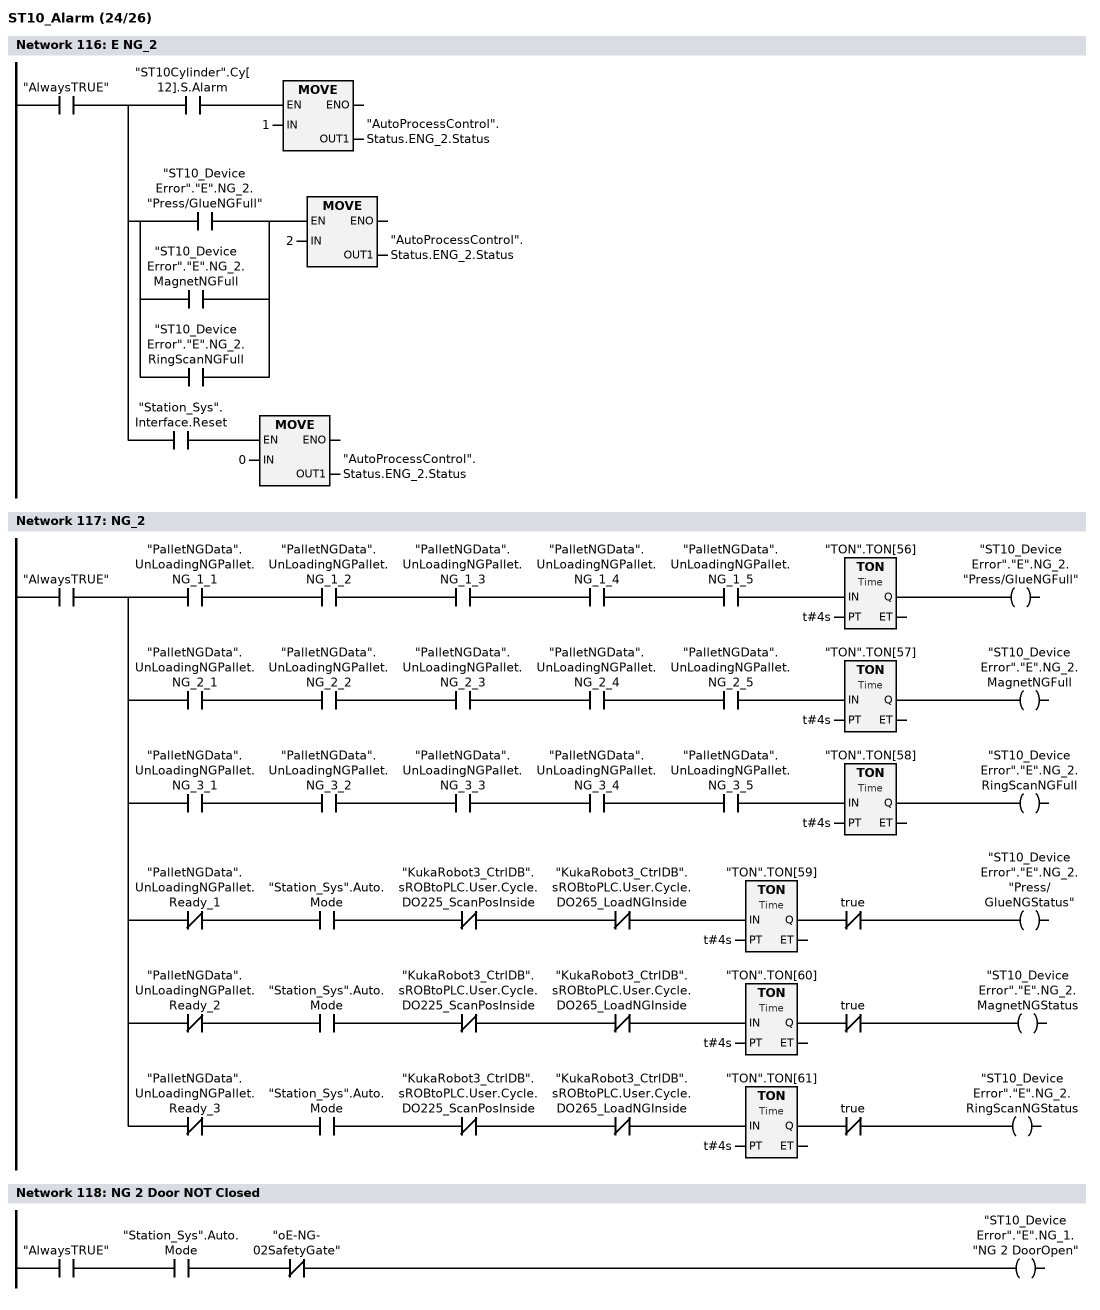
   RUNG wire#powerrail
      Contact( "AlwaysTRUE" )
      wire#w1
      Contact( "ST10Cylinder".Cy[12].S.Alarm )
      Move(in := 1, out1 => "AutoProcessControl".Status.ENG_2.Status)
   END_RUNG
   RUNG wire#w1
      Contact( "ST10_DeviceError"."E".NG_2."Press/GlueNGFull" )
      wire#w2
      Move(in := 2, out1 => "AutoProcessControl".Status.ENG_2.Status)
   END_RUNG
   RUNG wire#w1
      Contact( "ST10_DeviceError"."E".NG_2.MagnetNGFull )
   END_RUNG wire#w2
   RUNG wire#w1
      Contact( "ST10_DeviceError"."E".NG_2.RingScanNGFull )
   END_RUNG wire#w2
   RUNG wire#w1
      Contact( "Station_Sys".Interface.Reset )
      Move(in := 0, out1 => "AutoProcessControl".Status.ENG_2.Status)
   END_RUNG
   // the same network as SCL:
   IF "AlwaysTRUE" AND "ST10Cylinder".Cy[12].S.Alarm THEN
       "AutoProcessControl".Status.ENG_2.Status := 1;
   END_IF;
   IF "AlwaysTRUE" AND ("ST10_DeviceError"."E".NG_2."Press/GlueNGFull" OR "ST10_DeviceError"."E".NG_2.MagnetNGFull OR "ST10_DeviceError"."E".NG_2.RingScanNGFull) THEN
       "AutoProcessControl".Status.ENG_2.Status := 2;
   END_IF;
   IF "AlwaysTRUE" AND "Station_Sys".Interface.Reset THEN
       "AutoProcessControl".Status.ENG_2.Status := 0;
   END_IF;
END_REGION

REGION Network 117: NG_2
   RUNG wire#powerrail
      Contact( "AlwaysTRUE" )
      wire#w1
      Contact( "PalletNGData".UnLoadingNGPallet.NG_1_1 )
      Contact( "PalletNGData".UnLoadingNGPallet.NG_1_2 )
      Contact( "PalletNGData".UnLoadingNGPallet.NG_1_3 )
      Contact( "PalletNGData".UnLoadingNGPallet.NG_1_4 )
      Contact( "PalletNGData".UnLoadingNGPallet.NG_1_5 )
      { S7_Templates := "time_type := Time" } "TON".TON[56].TON(pt := t#4s, et =>)
      Coil( "ST10_DeviceError"."E".NG_2."Press/GlueNGFull" )
   END_RUNG
   RUNG wire#w1
      Contact( "PalletNGData".UnLoadingNGPallet.NG_2_1 )
      Contact( "PalletNGData".UnLoadingNGPallet.NG_2_2 )
      Contact( "PalletNGData".UnLoadingNGPallet.NG_2_3 )
      Contact( "PalletNGData".UnLoadingNGPallet.NG_2_4 )
      Contact( "PalletNGData".UnLoadingNGPallet.NG_2_5 )
      { S7_Templates := "time_type := Time" } "TON".TON[57].TON(pt := t#4s, et =>)
      Coil( "ST10_DeviceError"."E".NG_2.MagnetNGFull )
   END_RUNG
   RUNG wire#w1
      Contact( "PalletNGData".UnLoadingNGPallet.NG_3_1 )
      Contact( "PalletNGData".UnLoadingNGPallet.NG_3_2 )
      Contact( "PalletNGData".UnLoadingNGPallet.NG_3_3 )
      Contact( "PalletNGData".UnLoadingNGPallet.NG_3_4 )
      Contact( "PalletNGData".UnLoadingNGPallet.NG_3_5 )
      { S7_Templates := "time_type := Time" } "TON".TON[58].TON(pt := t#4s, et =>)
      Coil( "ST10_DeviceError"."E".NG_2.RingScanNGFull )
   END_RUNG
   RUNG wire#w1
      I_Contact( "PalletNGData".UnLoadingNGPallet.Ready_1 )
      Contact( "Station_Sys".Auto.Mode )
      I_Contact( "KukaRobot3_CtrlDB".sROBtoPLC.User.Cycle.DO225_ScanPosInside )
      I_Contact( "KukaRobot3_CtrlDB".sROBtoPLC.User.Cycle.DO265_LoadNGInside )
      { S7_Templates := "time_type := Time" } "TON".TON[59].TON(pt := t#4s, et =>)
      I_Contact( true )
      Coil( "ST10_DeviceError"."E".NG_2."Press/GlueNGStatus" )
   END_RUNG
   RUNG wire#w1
      I_Contact( "PalletNGData".UnLoadingNGPallet.Ready_2 )
      Contact( "Station_Sys".Auto.Mode )
      I_Contact( "KukaRobot3_CtrlDB".sROBtoPLC.User.Cycle.DO225_ScanPosInside )
      I_Contact( "KukaRobot3_CtrlDB".sROBtoPLC.User.Cycle.DO265_LoadNGInside )
      { S7_Templates := "time_type := Time" } "TON".TON[60].TON(pt := t#4s, et =>)
      I_Contact( true )
      Coil( "ST10_DeviceError"."E".NG_2.MagnetNGStatus )
   END_RUNG
   RUNG wire#w1
      I_Contact( "PalletNGData".UnLoadingNGPallet.Ready_3 )
      Contact( "Station_Sys".Auto.Mode )
      I_Contact( "KukaRobot3_CtrlDB".sROBtoPLC.User.Cycle.DO225_ScanPosInside )
      I_Contact( "KukaRobot3_CtrlDB".sROBtoPLC.User.Cycle.DO265_LoadNGInside )
      { S7_Templates := "time_type := Time" } "TON".TON[61].TON(pt := t#4s, et =>)
      I_Contact( true )
      Coil( "ST10_DeviceError"."E".NG_2.RingScanNGStatus )
   END_RUNG
   // the same network as SCL:
   "TON".TON[56].TON(IN := "AlwaysTRUE" AND "PalletNGData".UnLoadingNGPallet.NG_1_1 AND "PalletNGData".UnLoadingNGPallet.NG_1_2 AND "PalletNGData".UnLoadingNGPallet.NG_1_3 AND "PalletNGData".UnLoadingNGPallet.NG_1_4 AND "PalletNGData".UnLoadingNGPallet.NG_1_5,
                     PT := t#4s);
   "ST10_DeviceError"."E".NG_2."Press/GlueNGFull" := "TON".TON[56].Q;
   "TON".TON[57].TON(IN := "AlwaysTRUE" AND "PalletNGData".UnLoadingNGPallet.NG_2_1 AND "PalletNGData".UnLoadingNGPallet.NG_2_2 AND "PalletNGData".UnLoadingNGPallet.NG_2_3 AND "PalletNGData".UnLoadingNGPallet.NG_2_4 AND "PalletNGData".UnLoadingNGPallet.NG_2_5,
                     PT := t#4s);
   "ST10_DeviceError"."E".NG_2.MagnetNGFull := "TON".TON[57].Q;
   "TON".TON[58].TON(IN := "AlwaysTRUE" AND "PalletNGData".UnLoadingNGPallet.NG_3_1 AND "PalletNGData".UnLoadingNGPallet.NG_3_2 AND "PalletNGData".UnLoadingNGPallet.NG_3_3 AND "PalletNGData".UnLoadingNGPallet.NG_3_4 AND "PalletNGData".UnLoadingNGPallet.NG_3_5,
                     PT := t#4s);
   "ST10_DeviceError"."E".NG_2.RingScanNGFull := "TON".TON[58].Q;
   "TON".TON[59].TON(IN := "AlwaysTRUE" AND NOT "PalletNGData".UnLoadingNGPallet.Ready_1 AND "Station_Sys".Auto.Mode AND NOT "KukaRobot3_CtrlDB".sROBtoPLC.User.Cycle.DO225_ScanPosInside AND NOT "KukaRobot3_CtrlDB".sROBtoPLC.User.Cycle.DO265_LoadNGInside,
                     PT := t#4s);
   "ST10_DeviceError"."E".NG_2."Press/GlueNGStatus" := "TON".TON[59].Q AND NOT true;
   "TON".TON[60].TON(IN := "AlwaysTRUE" AND NOT "PalletNGData".UnLoadingNGPallet.Ready_2 AND "Station_Sys".Auto.Mode AND NOT "KukaRobot3_CtrlDB".sROBtoPLC.User.Cycle.DO225_ScanPosInside AND NOT "KukaRobot3_CtrlDB".sROBtoPLC.User.Cycle.DO265_LoadNGInside,
                     PT := t#4s);
   "ST10_DeviceError"."E".NG_2.MagnetNGStatus := "TON".TON[60].Q AND NOT true;
   "TON".TON[61].TON(IN := "AlwaysTRUE" AND NOT "PalletNGData".UnLoadingNGPallet.Ready_3 AND "Station_Sys".Auto.Mode AND NOT "KukaRobot3_CtrlDB".sROBtoPLC.User.Cycle.DO225_ScanPosInside AND NOT "KukaRobot3_CtrlDB".sROBtoPLC.User.Cycle.DO265_LoadNGInside,
                     PT := t#4s);
   "ST10_DeviceError"."E".NG_2.RingScanNGStatus := "TON".TON[61].Q AND NOT true;
END_REGION

REGION Network 118: NG 2 Door NOT Closed
   RUNG wire#powerrail
      Contact( "AlwaysTRUE" )
      Contact( "Station_Sys".Auto.Mode )
      I_Contact( "oE-NG-02SafetyGate" )
      Coil( "ST10_DeviceError"."E".NG_1."NG 2 DoorOpen" )
   END_RUNG
   // the same network as SCL:
   "ST10_DeviceError"."E".NG_1."NG 2 DoorOpen" := "AlwaysTRUE" AND "Station_Sys".Auto.Mode AND NOT "oE-NG-02SafetyGate";
END_REGION

REGION Network 119: Press1
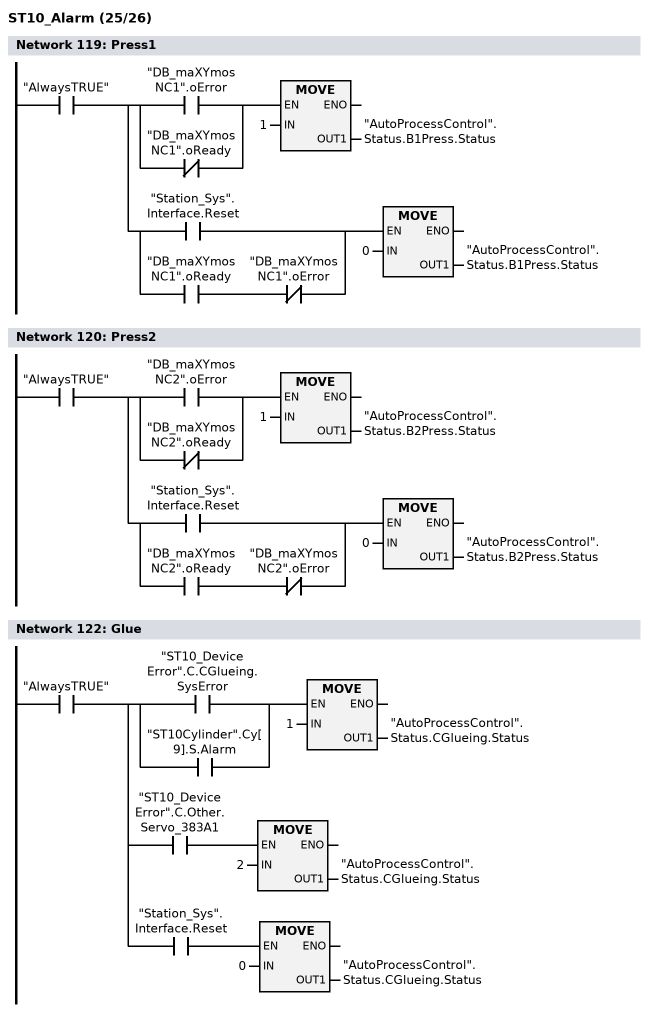
   RUNG wire#powerrail
      Contact( "AlwaysTRUE" )
      wire#w1
      Contact( "DB_maXYmosNC1".oError )
      wire#w2
      Move(in := 1, out1 => "AutoProcessControl".Status.B1Press.Status)
   END_RUNG
   RUNG wire#w1
      I_Contact( "DB_maXYmosNC1".oReady )
   END_RUNG wire#w2
   RUNG wire#w1
      Contact( "Station_Sys".Interface.Reset )
      wire#w3
      Move(in := 0, out1 => "AutoProcessControl".Status.B1Press.Status)
   END_RUNG
   RUNG wire#w1
      Contact( "DB_maXYmosNC1".oReady )
      I_Contact( "DB_maXYmosNC1".oError )
   END_RUNG wire#w3
   // the same network as SCL:
   IF "AlwaysTRUE" AND ("DB_maXYmosNC1".oError OR NOT "DB_maXYmosNC1".oReady) THEN
       "AutoProcessControl".Status.B1Press.Status := 1;
   END_IF;
   IF "AlwaysTRUE" AND ("Station_Sys".Interface.Reset OR ("DB_maXYmosNC1".oReady AND NOT "DB_maXYmosNC1".oError)) THEN
       "AutoProcessControl".Status.B1Press.Status := 0;
   END_IF;
END_REGION

REGION Network 120: Press2
   RUNG wire#powerrail
      Contact( "AlwaysTRUE" )
      wire#w1
      Contact( "DB_maXYmosNC2".oError )
      wire#w2
      Move(in := 1, out1 => "AutoProcessControl".Status.B2Press.Status)
   END_RUNG
   RUNG wire#w1
      I_Contact( "DB_maXYmosNC2".oReady )
   END_RUNG wire#w2
   RUNG wire#w1
      Contact( "Station_Sys".Interface.Reset )
      wire#w3
      Move(in := 0, out1 => "AutoProcessControl".Status.B2Press.Status)
   END_RUNG
   RUNG wire#w1
      Contact( "DB_maXYmosNC2".oReady )
      I_Contact( "DB_maXYmosNC2".oError )
   END_RUNG wire#w3
   // the same network as SCL:
   IF "AlwaysTRUE" AND ("DB_maXYmosNC2".oError OR NOT "DB_maXYmosNC2".oReady) THEN
       "AutoProcessControl".Status.B2Press.Status := 1;
   END_IF;
   IF "AlwaysTRUE" AND ("Station_Sys".Interface.Reset OR ("DB_maXYmosNC2".oReady AND NOT "DB_maXYmosNC2".oError)) THEN
       "AutoProcessControl".Status.B2Press.Status := 0;
   END_IF;
END_REGION

REGION Network 121: ******************** Glue ********************
END_REGION

REGION Network 122: Glue
   RUNG wire#powerrail
      Contact( "AlwaysTRUE" )
      wire#w1
      Contact( "ST10_DeviceError".C.CGlueing.SysError )
      wire#w2
      Move(in := 1, out1 => "AutoProcessControl".Status.CGlueing.Status)
   END_RUNG
   RUNG wire#w1
      Contact( "ST10Cylinder".Cy[9].S.Alarm )
   END_RUNG wire#w2
   RUNG wire#w1
      Contact( "ST10_DeviceError".C.Other.Servo_383A1 )
      Move(in := 2, out1 => "AutoProcessControl".Status.CGlueing.Status)
   END_RUNG
   RUNG wire#w1
      Contact( "Station_Sys".Interface.Reset )
      Move(in := 0, out1 => "AutoProcessControl".Status.CGlueing.Status)
   END_RUNG
   // the same network as SCL:
   IF "AlwaysTRUE" AND ("ST10_DeviceError".C.CGlueing.SysError OR "ST10Cylinder".Cy[9].S.Alarm) THEN
       "AutoProcessControl".Status.CGlueing.Status := 1;
   END_IF;
   IF "AlwaysTRUE" AND "ST10_DeviceError".C.Other.Servo_383A1 THEN
       "AutoProcessControl".Status.CGlueing.Status := 2;
   END_IF;
   IF "AlwaysTRUE" AND "Station_Sys".Interface.Reset THEN
       "AutoProcessControl".Status.CGlueing.Status := 0;
   END_IF;
END_REGION

REGION Network 123: A1 Table
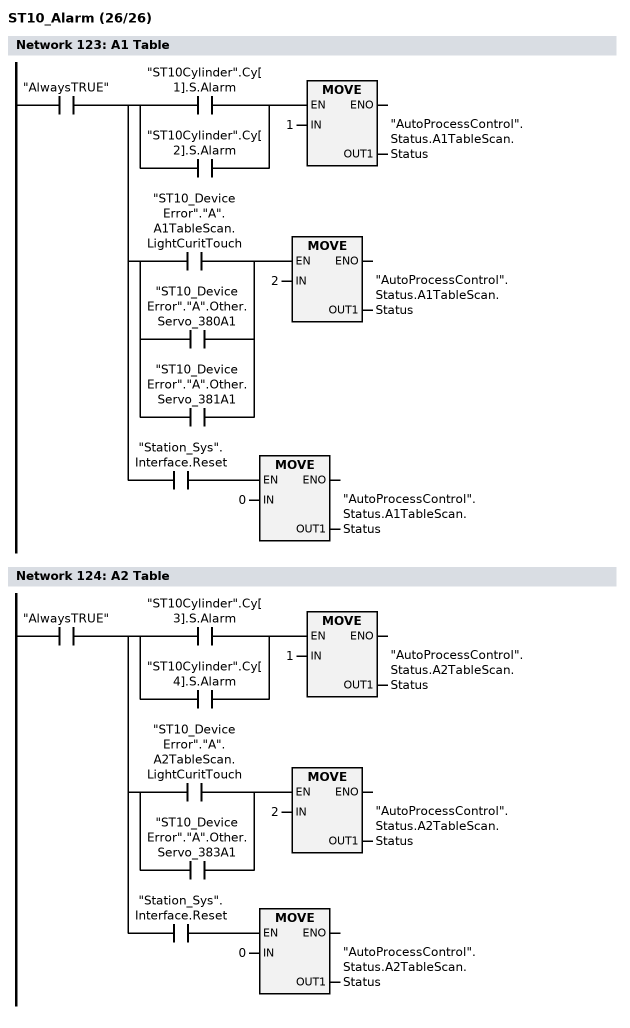
   RUNG wire#powerrail
      Contact( "AlwaysTRUE" )
      wire#w1
      Contact( "ST10Cylinder".Cy[1].S.Alarm )
      wire#w2
      Move(in := 1, out1 => "AutoProcessControl".Status.A1TableScan.Status)
   END_RUNG
   RUNG wire#w1
      Contact( "ST10Cylinder".Cy[2].S.Alarm )
   END_RUNG wire#w2
   RUNG wire#w1
      Contact( "ST10_DeviceError"."A".A1TableScan.LightCuritTouch )
      wire#w3
      Move(in := 2, out1 => "AutoProcessControl".Status.A1TableScan.Status)
   END_RUNG
   RUNG wire#w1
      Contact( "ST10_DeviceError"."A".Other.Servo_380A1 )
   END_RUNG wire#w3
   RUNG wire#w1
      Contact( "ST10_DeviceError"."A".Other.Servo_381A1 )
   END_RUNG wire#w3
   RUNG wire#w1
      Contact( "Station_Sys".Interface.Reset )
      Move(in := 0, out1 => "AutoProcessControl".Status.A1TableScan.Status)
   END_RUNG
   // the same network as SCL:
   IF "AlwaysTRUE" AND ("ST10Cylinder".Cy[1].S.Alarm OR "ST10Cylinder".Cy[2].S.Alarm) THEN
       "AutoProcessControl".Status.A1TableScan.Status := 1;
   END_IF;
   IF "AlwaysTRUE" AND ("ST10_DeviceError"."A".A1TableScan.LightCuritTouch OR "ST10_DeviceError"."A".Other.Servo_380A1 OR "ST10_DeviceError"."A".Other.Servo_381A1) THEN
       "AutoProcessControl".Status.A1TableScan.Status := 2;
   END_IF;
   IF "AlwaysTRUE" AND "Station_Sys".Interface.Reset THEN
       "AutoProcessControl".Status.A1TableScan.Status := 0;
   END_IF;
END_REGION

REGION Network 124: A2 Table
   RUNG wire#powerrail
      Contact( "AlwaysTRUE" )
      wire#w1
      Contact( "ST10Cylinder".Cy[3].S.Alarm )
      wire#w2
      Move(in := 1, out1 => "AutoProcessControl".Status.A2TableScan.Status)
   END_RUNG
   RUNG wire#w1
      Contact( "ST10Cylinder".Cy[4].S.Alarm )
   END_RUNG wire#w2
   RUNG wire#w1
      Contact( "ST10_DeviceError"."A".A2TableScan.LightCuritTouch )
      wire#w3
      Move(in := 2, out1 => "AutoProcessControl".Status.A2TableScan.Status)
   END_RUNG
   RUNG wire#w1
      Contact( "ST10_DeviceError"."A".Other.Servo_383A1 )
   END_RUNG wire#w3
   RUNG wire#w1
      Contact( "Station_Sys".Interface.Reset )
      Move(in := 0, out1 => "AutoProcessControl".Status.A2TableScan.Status)
   END_RUNG
   // the same network as SCL:
   IF "AlwaysTRUE" AND ("ST10Cylinder".Cy[3].S.Alarm OR "ST10Cylinder".Cy[4].S.Alarm) THEN
       "AutoProcessControl".Status.A2TableScan.Status := 1;
   END_IF;
   IF "AlwaysTRUE" AND ("ST10_DeviceError"."A".A2TableScan.LightCuritTouch OR "ST10_DeviceError"."A".Other.Servo_383A1) THEN
       "AutoProcessControl".Status.A2TableScan.Status := 2;
   END_IF;
   IF "AlwaysTRUE" AND "Station_Sys".Interface.Reset THEN
       "AutoProcessControl".Status.A2TableScan.Status := 0;
   END_IF;
END_REGION
END_FUNCTION

FUNCTION "CheckData" : Void   // FC4023, SCL
{ S7_Optimized_Access := 'FALSE' }
// stored: AutoNumber false, SetENOAutomatically false
   VAR_INPUT
      DBNo : Int;
      DBBNO : Int;
      ByteLenth : Int;
   END_VAR
   VAR_OUTPUT
      AlarmON : Bool;
   END_VAR
   VAR_TEMP
      AlarmByte : Int;
      tByte : Int;
   END_VAR
BEGIN
   #AlarmON := 0;
   #AlarmByte := 0;
   IF #ByteLenth>0 THEN
       FOR #tByte:=0 TO #ByteLenth-1 DO
           IF PEEK_BYTE(area:=16#84,dbNumber:=#DBNo,byteOffset:=#DBBNO+#tByte)<>0 THEN
               #AlarmON := TRUE;
               #AlarmByte := #DBBNO + #tByte;
               EXIT;
           ELSE
               #AlarmON := false;
               #AlarmByte := 0;
           END_IF;
       END_FOR;
   END_IF;
END_FUNCTION

FUNCTION "ST10_Warning" : Void   // FC1006, LAD
{ S7_Optimized_Access := 'FALSE' }
// stored: AutoNumber false, SetENOAutomatically false
   VAR_TEMP
      tpAlwayoff : Bool;
   END_VAR
BEGIN

REGION Network 1
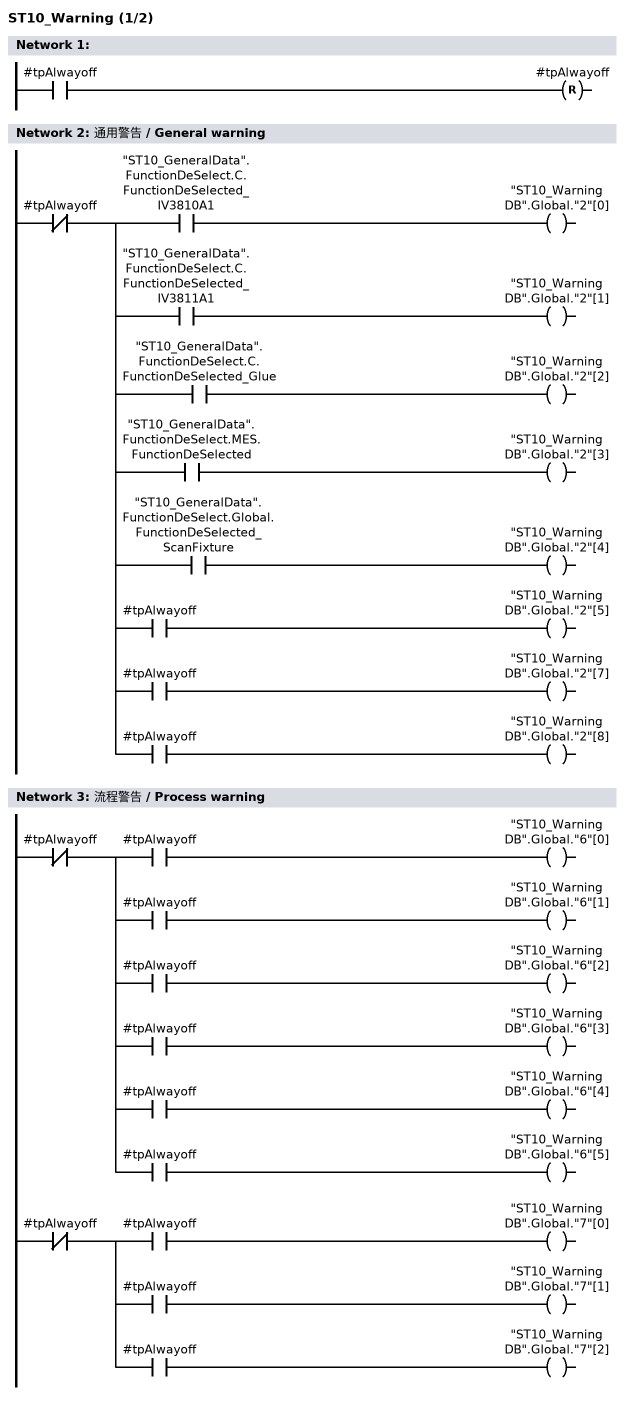
   RUNG wire#powerrail
      Contact( #tpAlwayoff )
      R_Coil( #tpAlwayoff )
   END_RUNG
   // the same network as SCL:
   IF #tpAlwayoff THEN #tpAlwayoff := FALSE; END_IF;
END_REGION

REGION Network 2: 通用警告 / General warning
   RUNG wire#powerrail
      I_Contact( #tpAlwayoff )
      wire#w1
      Contact( "ST10_GeneralData".FunctionDeSelect.C.FunctionDeSelected_IV3810A1 )
      Coil( "ST10_WarningDB".Global."2"[0] )
   END_RUNG
   RUNG wire#w1
      Contact( "ST10_GeneralData".FunctionDeSelect.C.FunctionDeSelected_IV3811A1 )
      Coil( "ST10_WarningDB".Global."2"[1] )
   END_RUNG
   RUNG wire#w1
      Contact( "ST10_GeneralData".FunctionDeSelect.C.FunctionDeSelected_Glue )
      Coil( "ST10_WarningDB".Global."2"[2] )
   END_RUNG
   RUNG wire#w1
      Contact( "ST10_GeneralData".FunctionDeSelect.MES.FunctionDeSelected )
      Coil( "ST10_WarningDB".Global."2"[3] )
   END_RUNG
   RUNG wire#w1
      Contact( "ST10_GeneralData".FunctionDeSelect.Global.FunctionDeSelected_ScanFixture )
      Coil( "ST10_WarningDB".Global."2"[4] )
   END_RUNG
   RUNG wire#w1
      Contact( #tpAlwayoff )
      Coil( "ST10_WarningDB".Global."2"[5] )
   END_RUNG
   RUNG wire#w1
      Contact( #tpAlwayoff )
      Coil( "ST10_WarningDB".Global."2"[7] )
   END_RUNG
   RUNG wire#w1
      Contact( #tpAlwayoff )
      Coil( "ST10_WarningDB".Global."2"[8] )
   END_RUNG
   // the same network as SCL:
   "ST10_WarningDB".Global."2"[0] := NOT #tpAlwayoff AND "ST10_GeneralData".FunctionDeSelect.C.FunctionDeSelected_IV3810A1;
   "ST10_WarningDB".Global."2"[1] := NOT #tpAlwayoff AND "ST10_GeneralData".FunctionDeSelect.C.FunctionDeSelected_IV3811A1;
   "ST10_WarningDB".Global."2"[2] := NOT #tpAlwayoff AND "ST10_GeneralData".FunctionDeSelect.C.FunctionDeSelected_Glue;
   "ST10_WarningDB".Global."2"[3] := NOT #tpAlwayoff AND "ST10_GeneralData".FunctionDeSelect.MES.FunctionDeSelected;
   "ST10_WarningDB".Global."2"[4] := NOT #tpAlwayoff AND "ST10_GeneralData".FunctionDeSelect.Global.FunctionDeSelected_ScanFixture;
   "ST10_WarningDB".Global."2"[5] := NOT #tpAlwayoff AND #tpAlwayoff;
   "ST10_WarningDB".Global."2"[7] := NOT #tpAlwayoff AND #tpAlwayoff;
   "ST10_WarningDB".Global."2"[8] := NOT #tpAlwayoff AND #tpAlwayoff;
END_REGION

REGION Network 3: 流程警告 / Process warning
   RUNG wire#powerrail
      I_Contact( #tpAlwayoff )
      wire#w1
      Contact( #tpAlwayoff )
      Coil( "ST10_WarningDB".Global."6"[0] )
   END_RUNG
   RUNG wire#w1
      Contact( #tpAlwayoff )
      Coil( "ST10_WarningDB".Global."6"[1] )
   END_RUNG
   RUNG wire#w1
      Contact( #tpAlwayoff )
      Coil( "ST10_WarningDB".Global."6"[2] )
   END_RUNG
   RUNG wire#w1
      Contact( #tpAlwayoff )
      Coil( "ST10_WarningDB".Global."6"[3] )
   END_RUNG
   RUNG wire#w1
      Contact( #tpAlwayoff )
      Coil( "ST10_WarningDB".Global."6"[4] )
   END_RUNG
   RUNG wire#w1
      Contact( #tpAlwayoff )
      Coil( "ST10_WarningDB".Global."6"[5] )
   END_RUNG
   RUNG wire#powerrail
      I_Contact( #tpAlwayoff )
      wire#w2
      Contact( #tpAlwayoff )
      Coil( "ST10_WarningDB".Global."7"[0] )
   END_RUNG
   RUNG wire#w2
      Contact( #tpAlwayoff )
      Coil( "ST10_WarningDB".Global."7"[1] )
   END_RUNG
   RUNG wire#w2
      Contact( #tpAlwayoff )
      Coil( "ST10_WarningDB".Global."7"[2] )
   END_RUNG
   // the same network as SCL:
   "ST10_WarningDB".Global."6"[0] := NOT #tpAlwayoff AND #tpAlwayoff;
   "ST10_WarningDB".Global."6"[1] := NOT #tpAlwayoff AND #tpAlwayoff;
   "ST10_WarningDB".Global."6"[2] := NOT #tpAlwayoff AND #tpAlwayoff;
   "ST10_WarningDB".Global."6"[3] := NOT #tpAlwayoff AND #tpAlwayoff;
   "ST10_WarningDB".Global."6"[4] := NOT #tpAlwayoff AND #tpAlwayoff;
   "ST10_WarningDB".Global."6"[5] := NOT #tpAlwayoff AND #tpAlwayoff;
   "ST10_WarningDB".Global."7"[0] := NOT #tpAlwayoff AND #tpAlwayoff;
   "ST10_WarningDB".Global."7"[1] := NOT #tpAlwayoff AND #tpAlwayoff;
   "ST10_WarningDB".Global."7"[2] := NOT #tpAlwayoff AND #tpAlwayoff;
END_REGION

REGION Network 4: 标定警告 / Calibration warning
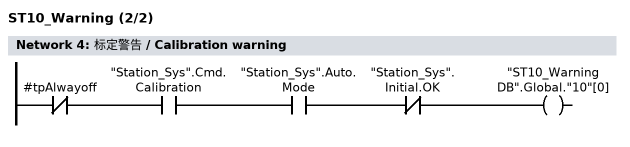
   RUNG wire#powerrail
      I_Contact( #tpAlwayoff )
      Contact( "Station_Sys".Cmd.Calibration )
      Contact( "Station_Sys".Auto.Mode )
      I_Contact( "Station_Sys".Initial.OK )
      Coil( "ST10_WarningDB".Global."10"[0] )
   END_RUNG
   // the same network as SCL:
   "ST10_WarningDB".Global."10"[0] := NOT #tpAlwayoff AND "Station_Sys".Cmd.Calibration AND "Station_Sys".Auto.Mode AND NOT "Station_Sys".Initial.OK;
END_REGION
END_FUNCTION

FUNCTION "ST10_Tip" : Void   // FC1007, LAD
{ S7_Optimized_Access := 'FALSE' }
// stored: AutoNumber false, SetENOAutomatically false
   VAR_TEMP   // added for the SCL form of the ladder/FBD networks
      _w1 : Bool;
   END_VAR
BEGIN

NETWORK
TITLE = Gloal Tips

//7000: 设备未上电，请先按下复位按钮，在按下控制开按钮
//      AN    "iHMIE-StopPB"
//     AN    "iE_StopPB_1"
//     AN    "iE_StopPB_2"
//     AN    "iE_StopPB_3"
//     AN    "ST350_Sys".Status.ControlOn
//     =     "ST350_TipDB".Global."1".ControlOn

//7001：设备存在故障，请查看报警信息，消除故障，然后按复位按钮
//     A     "ST350_Sys".Status.ControlOn
//     O(
//      A     "iHMIE-StopPB"
//     O     "iE_StopPB_1"
//     O     "iE_StopPB_2"
//     O     "iE_StopPB_3"
//    )
//    A     "ST350_Sys".Alarm.ON
//    =     "ST350_TipDB".Global."1".Reset

//7002: 未选择配方，请在换型页面选择配方
//      A     "ST350_Sys".Status.ControlOn
//     AN    "ST350_TipDB".Global."1".Reset
//
//      AN    "ST350_RecipeDB".Recipe.Equal
//     =     "ST350_TipDB".Global."2"[0]

//7003:设备未选择自动，请选择自动模式
//      A     "ST350_Sys".Status.ControlOn
//     AN    "ST350_TipDB".Global."1".Reset
//     A     "ST350_RecipeDB".Recipe.Equal
//     AN    "ST350_Sys".Interface.Auto.Mode

//    =     "ST350_TipDB".Global."1".SelectAutoMode

//7004:设备初始化，请启动设备初始化
//     A     "ST350_Sys".Status.ControlOn
//     AN    "ST350_TipDB".Global."1".Reset
//      A     "ST350_RecipeDB".Recipe.Equal
//     A     "ST350_Sys".Interface.Auto.Mode

//    AN    "ST350_Sys".Initial.OK
//     =     "ST350_TipDB".Global."2"[1]


//7005:设备未启动，请启动自动运行
//     A     "ST350_Sys".Status.ControlOn
//    AN    "ST350_TipDB".Global."1".Reset
//    A     "ST350_RecipeDB".Recipe.Equal
//    A     "ST350_Sys".Interface.Auto.Mode
//    A     "ST350_Sys".Initial.OK
//
//    AN    "ST350_Sys".Interface.Auto.Running
//    AN    "ST350_Sys".Interface.Auto.AllRun
//    =     "ST350_TipDB".Global."1".AutoModeRunning

REGION Network 2: Gloal Tips:7000: 设备未上电，请先按下复位按钮，在按下控制开按钮 / Gloal Tips:7000: The device is not powered on, please press the reset button first, and then press the control button
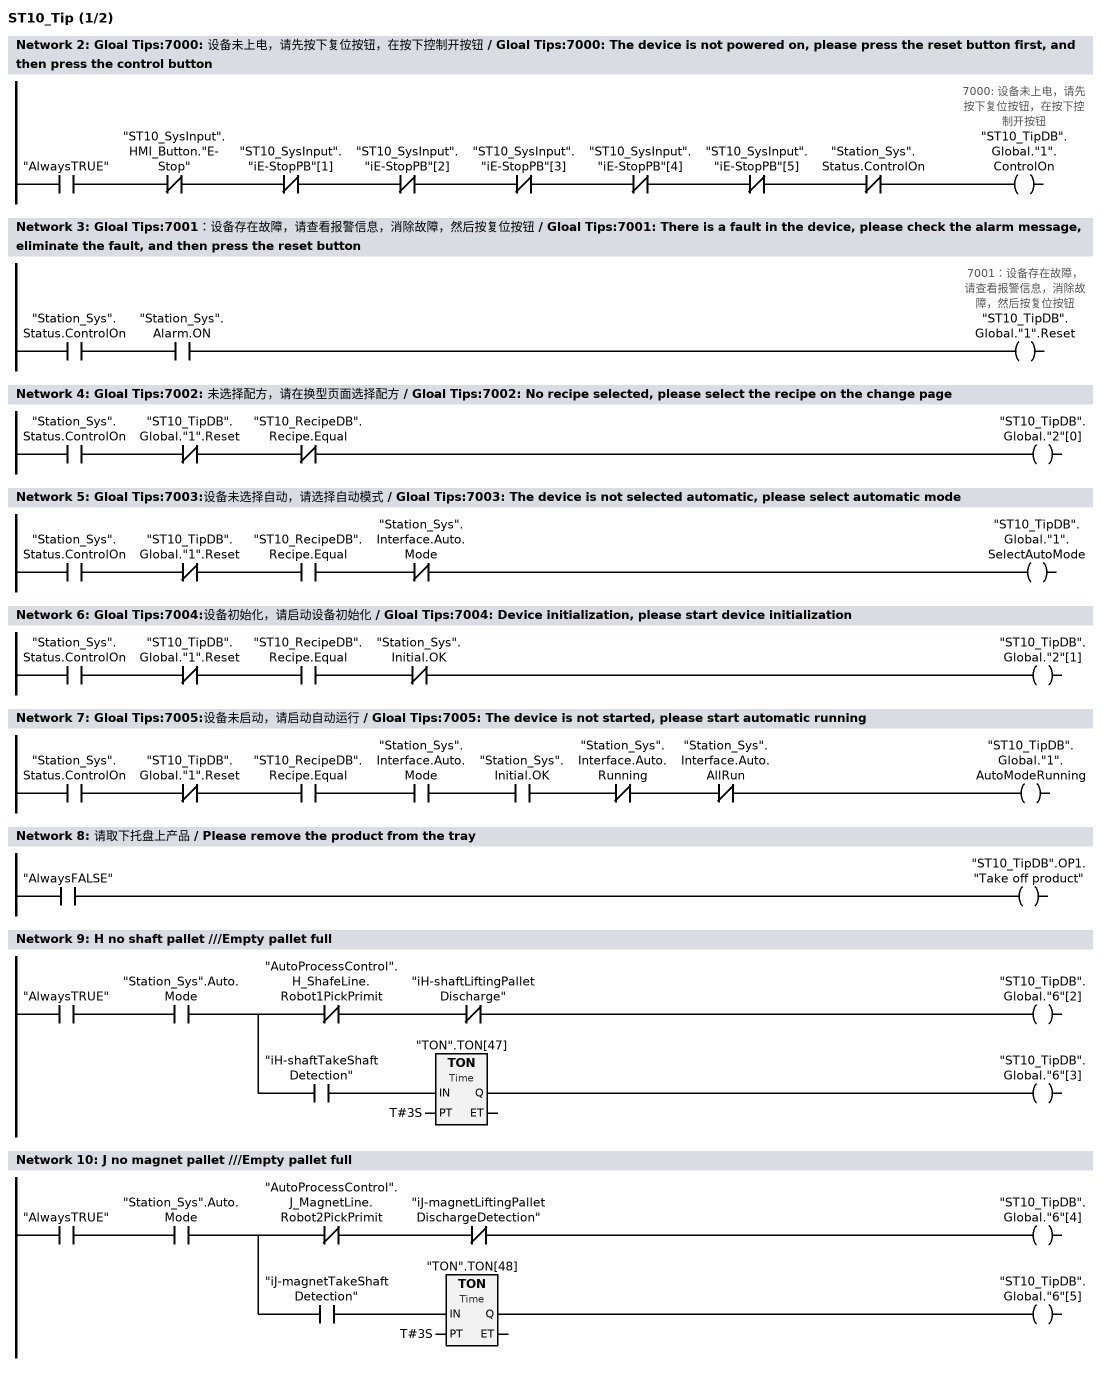
   RUNG wire#powerrail
      Contact( "AlwaysTRUE" )
      I_Contact( "ST10_SysInput".HMI_Button."E-Stop" )
      I_Contact( "ST10_SysInput"."iE-StopPB"[1] )
      I_Contact( "ST10_SysInput"."iE-StopPB"[2] )
      I_Contact( "ST10_SysInput"."iE-StopPB"[3] )
      I_Contact( "ST10_SysInput"."iE-StopPB"[4] )
      I_Contact( "ST10_SysInput"."iE-StopPB"[5] )
      I_Contact( "Station_Sys".Status.ControlOn )
      Coil( "ST10_TipDB".Global."1".ControlOn )   // 7000: 设备未上电，请先按下复位按钮，在按下控制开按钮
   END_RUNG
   // the same network as SCL:
   "ST10_TipDB".Global."1".ControlOn := "AlwaysTRUE" AND NOT "ST10_SysInput".HMI_Button."E-Stop" AND NOT "ST10_SysInput"."iE-StopPB"[1] AND NOT "ST10_SysInput"."iE-StopPB"[2] AND NOT "ST10_SysInput"."iE-StopPB"[3] AND NOT "ST10_SysInput"."iE-StopPB"[4] AND NOT "ST10_SysInput"."iE-StopPB"[5] AND NOT "Station_Sys".Status.ControlOn;   // 7000: 设备未上电，请先按下复位按钮，在按下控制开按钮
END_REGION

REGION Network 3: Gloal Tips:7001：设备存在故障，请查看报警信息，消除故障，然后按复位按钮 / Gloal Tips:7001: There is a fault in the device, please check the alarm message, eliminate the fault, and then press the reset button
   RUNG wire#powerrail
      Contact( "Station_Sys".Status.ControlOn )
      Contact( "Station_Sys".Alarm.ON )
      Coil( "ST10_TipDB".Global."1".Reset )   // 7001：设备存在故障，请查看报警信息，消除故障，然后按复位按钮
   END_RUNG
   // the same network as SCL:
   "ST10_TipDB".Global."1".Reset := "Station_Sys".Status.ControlOn AND "Station_Sys".Alarm.ON;   // 7001：设备存在故障，请查看报警信息，消除故障，然后按复位按钮
END_REGION

REGION Network 4: Gloal Tips:7002: 未选择配方，请在换型页面选择配方 / Gloal Tips:7002: No recipe selected, please select the recipe on the change page
   RUNG wire#powerrail
      Contact( "Station_Sys".Status.ControlOn )
      I_Contact( "ST10_TipDB".Global."1".Reset )
      I_Contact( "ST10_RecipeDB".Recipe.Equal )
      Coil( "ST10_TipDB".Global."2"[0] )
   END_RUNG
   // the same network as SCL:
   "ST10_TipDB".Global."2"[0] := "Station_Sys".Status.ControlOn AND NOT "ST10_TipDB".Global."1".Reset AND NOT "ST10_RecipeDB".Recipe.Equal;
END_REGION

REGION Network 5: Gloal Tips:7003:设备未选择自动，请选择自动模式 / Gloal Tips:7003: The device is not selected automatic, please select automatic mode
   RUNG wire#powerrail
      Contact( "Station_Sys".Status.ControlOn )
      I_Contact( "ST10_TipDB".Global."1".Reset )
      Contact( "ST10_RecipeDB".Recipe.Equal )
      I_Contact( "Station_Sys".Interface.Auto.Mode )
      Coil( "ST10_TipDB".Global."1".SelectAutoMode )
   END_RUNG
   // the same network as SCL:
   "ST10_TipDB".Global."1".SelectAutoMode := "Station_Sys".Status.ControlOn AND NOT "ST10_TipDB".Global."1".Reset AND "ST10_RecipeDB".Recipe.Equal AND NOT "Station_Sys".Interface.Auto.Mode;
END_REGION

REGION Network 6: Gloal Tips:7004:设备初始化，请启动设备初始化 / Gloal Tips:7004: Device initialization, please start device initialization
   RUNG wire#powerrail
      Contact( "Station_Sys".Status.ControlOn )
      I_Contact( "ST10_TipDB".Global."1".Reset )
      Contact( "ST10_RecipeDB".Recipe.Equal )
      I_Contact( "Station_Sys".Initial.OK )
      Coil( "ST10_TipDB".Global."2"[1] )
   END_RUNG
   // the same network as SCL:
   "ST10_TipDB".Global."2"[1] := "Station_Sys".Status.ControlOn AND NOT "ST10_TipDB".Global."1".Reset AND "ST10_RecipeDB".Recipe.Equal AND NOT "Station_Sys".Initial.OK;
END_REGION

REGION Network 7: Gloal Tips:7005:设备未启动，请启动自动运行 / Gloal Tips:7005: The device is not started, please start automatic running
   RUNG wire#powerrail
      Contact( "Station_Sys".Status.ControlOn )
      I_Contact( "ST10_TipDB".Global."1".Reset )
      Contact( "ST10_RecipeDB".Recipe.Equal )
      Contact( "Station_Sys".Interface.Auto.Mode )
      Contact( "Station_Sys".Initial.OK )
      I_Contact( "Station_Sys".Interface.Auto.Running )
      I_Contact( "Station_Sys".Interface.Auto.AllRun )
      Coil( "ST10_TipDB".Global."1".AutoModeRunning )
   END_RUNG
   // the same network as SCL:
   "ST10_TipDB".Global."1".AutoModeRunning := "Station_Sys".Status.ControlOn AND NOT "ST10_TipDB".Global."1".Reset AND "ST10_RecipeDB".Recipe.Equal AND "Station_Sys".Interface.Auto.Mode AND "Station_Sys".Initial.OK AND NOT "Station_Sys".Interface.Auto.Running AND NOT "Station_Sys".Interface.Auto.AllRun;
END_REGION

REGION Network 8: 请取下托盘上产品 / Please remove the product from the tray
   RUNG wire#powerrail
      Contact( "AlwaysFALSE" )
      Coil( "ST10_TipDB".OP1."Take off product" )
   END_RUNG
   // the same network as SCL:
   "ST10_TipDB".OP1."Take off product" := "AlwaysFALSE";
END_REGION

REGION Network 9: H no shaft pallet ///Empty pallet full
   RUNG wire#powerrail
      Contact( "AlwaysTRUE" )
      Contact( "Station_Sys".Auto.Mode )
      wire#w1
      I_Contact( "AutoProcessControl".H_ShafeLine.Robot1PickPrimit )
      I_Contact( "iH-shaftLiftingPalletDischarge" )
      Coil( "ST10_TipDB".Global."6"[2] )
   END_RUNG
   RUNG wire#w1
      Contact( "iH-shaftTakeShaftDetection" )
      { S7_Templates := "time_type := Time" } "TON".TON[47].TON(pt := T#3S, et =>)
      Coil( "ST10_TipDB".Global."6"[3] )
   END_RUNG
   // the same network as SCL:
   #_w1 := "AlwaysTRUE" AND "Station_Sys".Auto.Mode;
   "ST10_TipDB".Global."6"[2] := #_w1 AND NOT "AutoProcessControl".H_ShafeLine.Robot1PickPrimit AND NOT "iH-shaftLiftingPalletDischarge";
   "TON".TON[47].TON(IN := #_w1 AND "iH-shaftTakeShaftDetection", PT := T#3S);
   "ST10_TipDB".Global."6"[3] := "TON".TON[47].Q;
END_REGION

REGION Network 10: J no magnet pallet ///Empty pallet full
   RUNG wire#powerrail
      Contact( "AlwaysTRUE" )
      Contact( "Station_Sys".Auto.Mode )
      wire#w1
      I_Contact( "AutoProcessControl".J_MagnetLine.Robot2PickPrimit )
      I_Contact( "iJ-magnetLiftingPalletDischargeDetection" )
      Coil( "ST10_TipDB".Global."6"[4] )
   END_RUNG
   RUNG wire#w1
      Contact( "iJ-magnetTakeShaftDetection" )
      { S7_Templates := "time_type := Time" } "TON".TON[48].TON(pt := T#3S, et =>)
      Coil( "ST10_TipDB".Global."6"[5] )
   END_RUNG
   // the same network as SCL:
   #_w1 := "AlwaysTRUE" AND "Station_Sys".Auto.Mode;
   "ST10_TipDB".Global."6"[4] := #_w1 AND NOT "AutoProcessControl".J_MagnetLine.Robot2PickPrimit AND NOT "iJ-magnetLiftingPalletDischargeDetection";
   "TON".TON[48].TON(IN := #_w1 AND "iJ-magnetTakeShaftDetection", PT := T#3S);
   "ST10_TipDB".Global."6"[5] := "TON".TON[48].Q;
END_REGION

REGION Network 11: K no magnet pallet ///Empty pallet full
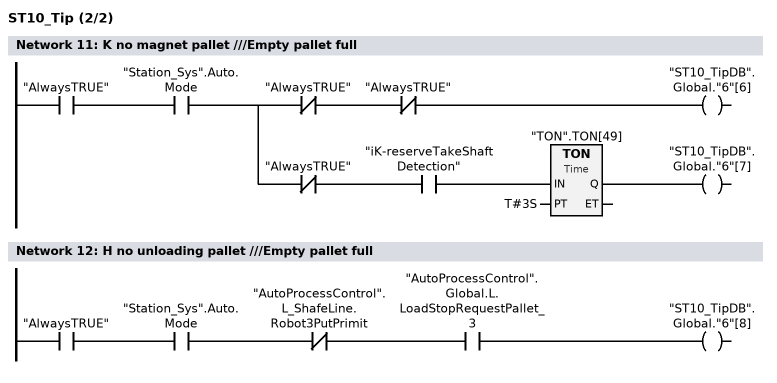
   RUNG wire#powerrail
      Contact( "AlwaysTRUE" )
      Contact( "Station_Sys".Auto.Mode )
      wire#w1
      I_Contact( "AlwaysTRUE" )
      I_Contact( "AlwaysTRUE" )
      Coil( "ST10_TipDB".Global."6"[6] )
   END_RUNG
   RUNG wire#w1
      I_Contact( "AlwaysTRUE" )
      Contact( "iK-reserveTakeShaftDetection" )
      { S7_Templates := "time_type := Time" } "TON".TON[49].TON(pt := T#3S, et =>)
      Coil( "ST10_TipDB".Global."6"[7] )
   END_RUNG
   // the same network as SCL:
   #_w1 := "AlwaysTRUE" AND "Station_Sys".Auto.Mode;
   "ST10_TipDB".Global."6"[6] := #_w1 AND NOT "AlwaysTRUE" AND NOT "AlwaysTRUE";
   "TON".TON[49].TON(IN := #_w1 AND NOT "AlwaysTRUE" AND "iK-reserveTakeShaftDetection", PT := T#3S);
   "ST10_TipDB".Global."6"[7] := "TON".TON[49].Q;
END_REGION

REGION Network 12: H no unloading pallet ///Empty pallet full
   RUNG wire#powerrail
      Contact( "AlwaysTRUE" )
      Contact( "Station_Sys".Auto.Mode )
      I_Contact( "AutoProcessControl".L_ShafeLine.Robot3PutPrimit )
      Contact( "AutoProcessControl".Global.L.LoadStopRequestPallet_3 )
      Coil( "ST10_TipDB".Global."6"[8] )
   END_RUNG
   // the same network as SCL:
   "ST10_TipDB".Global."6"[8] := "AlwaysTRUE" AND "Station_Sys".Auto.Mode AND NOT "AutoProcessControl".L_ShafeLine.Robot3PutPrimit AND "AutoProcessControl".Global.L.LoadStopRequestPallet_3;
END_REGION
END_FUNCTION

FUNCTION "CylinderCtrl_V2" : Void   // FC3011, SCL
TITLE = CylinderV3
{ S7_Optimized_Access := 'FALSE' }
AUTHOR : JM
FAMILY : RCS
VERSION : 18.2
// this function is only used for cylinder control
// stored: AutoNumber false, IsIECCheckEnabled false, SetENOAutomatically true, UDAEnableTagReadback false
   VAR_INPUT
      iReset : Bool;   // reset action
      iRun : Bool;   // system run
      iEStop : Bool;   // e_stop monitor
      iManualMode : Bool;   // manual mode
      iAutoMode : Bool;   // auto mode
      iEnableAlarm : Bool;   // alarm will popup up
      iPulse100mS : Bool;   // pulse *100ms
      iPulse1S : Bool;   // pulse*1s
      iCyDBNO : Word;   // Interface data block number
      iCyCounts : Int;   // total counts of cylinder to be used[must be>=1 and <=100]
      iDevAlarmDBNum : Word;   // Device Alarm DataBlock Alarm
   END_VAR
   VAR_TEMP
      CyInterface : "Cyl";
      CyRany : Any;
      cyRSany AT CyRany : Struct
         SyntaxID : Byte;
         DataType : Byte;
         RepetitionFactor : Int;
         DB_Number : Word;
         MemoryAreaAddress : DWord;
      END_STRUCT;
      CyDany : Any;
      CyDSany AT CyDany : Struct
         SyntaxID : Byte;
         DataType : Byte;
         RepetitionFactor : Int;
         DB_Number : Word;
         MemoryAreaAddress : DWord;
      END_STRUCT;
      tpCounts : Int;
      tpi : Int;
      tpRetVal : Int;
   END_VAR
BEGIN
   //---------------------------------------------------------------//
   //FunctionName:CylinderV3
   //FunctionDescription:Cylinder Control block
   //---------------------------------------------------------------//
   (*in:

   #iReset  Bool            reset action
   #iRun    Bool            system run
   #iE_stop Bool            e_stop monitor
   #iManualMode Bool        manual mode
   #iAutoMode   Bool        auto mode
   #iEnableAlarm    Bool        alarm will popup up
   #iPulse_100mS    Bool        pulse *100ms
   iPulse_1S   Bool        pulse*1s
   iCyDBNO Int Int     Interface data block number
   iCyCounts   Int     total counts OF "Cylinder" TO be used[must be>=1 AND <=100]

   //inout:
   //out:
   *)
   //---------------------------------------------------------------//
   //Version:V3
   //D&T:2016-11-14
   //Group:RCS
   //Author:JiangMing
   //-------------------------Modify1----------------------------------//
   //Version:
   //D&T:2016-11-17
   //Group: RCS
   //Author:JiangMing
   //Modify:Update cylinder no as output interface
   //-------------------------Modify2----------------------------------//
   //Version:       V18.3
   //D&T:           2020-06-11
   //Group:         RCS
   //Author:        JM
   //Modify:        1.MaxCylinder count 200 
   //               2.Refine alarm interface
   IF #iCyCounts > 200 THEN
       #tpCounts := 200;
   ELSE
       #tpCounts := #iCyCounts;
   END_IF;
   //input

   FOR #tpi := 0 TO #tpCounts-1 DO
       //****************************************************************************************//
       #cyRSany.SyntaxID := 16#10;
       #cyRSany.DataType := 16#02;
       #cyRSany.RepetitionFactor := 22;
       #cyRSany.DB_Number := #iCyDBNO;
       #cyRSany.MemoryAreaAddress := 16#8400_0000 OR (SHL(IN := INT_TO_DWORD(#tpi * 22), N := 3));///
       //-----------------------------//
       #CyDSany.SyntaxID := 16#10;
       #CyDSany.DataType := 16#02;
       #CyDSany.RepetitionFactor := 22;
       #CyDSany.DB_Number := 0;
       #CyDSany.MemoryAreaAddress := 16#8700_0000 OR (SHL(IN := INT_TO_DWORD(0), N := 3));///
       #tpRetVal := BLKMOV(SRCBLK := #CyRany, DSTBLK => #CyDany);
       //***************************************************************************************//
       "CylinderModule_V2"(iReset := #iReset,
                        iRun := #iRun,
                        iEStop := #iEStop,
                        iManualMode := #iManualMode,
                        iAutoMode := #iAutoMode,
                        iEnableAlarm := #iEnableAlarm,
                        iPulse100mS := #iPulse100mS,
                        iPulse1S := #iPulse1S,
                        iError := #CyInterface.In.Error,
                        iGoWorkInterlock := #CyInterface.In.GoWorkInterlock,
                        iGoHomeInterlock := #CyInterface.In.GoHomeInterlock,
                        iWorkPositionSensor := #CyInterface.In.WorkPositionSensor,
                        iHomePositionSensor := #CyInterface.In.HomePositionSensor,
                        iValveType := #CyInterface.In.ValveType,
                        iManualOutputType := #CyInterface.In.ManualOutputType,
                        iFaultTime := #CyInterface.In.FaultTime,
                        iOnPositionTime := #CyInterface.In.OnPositionTime,
                           ioResetOut:=#CyInterface.Inout.ResetOut,
                        ioGoWorkPosition := #CyInterface.Out.GoWorkPosition,
                        ioGoHomePosition := #CyInterface.Out.GoHomePosition,
                        oGoWP_ButtonActive => #CyInterface.Out.GoWPButtonActive,
                        oGoHP_ButtonActive => #CyInterface.Out.GoHPButtonActive,
                        ioGoWorkFault := #CyInterface.Out.GoWorkFault,
                        ioGoHomeFault := #CyInterface.Out.GoHomeFault,
                        ioSensorPositionFault := #CyInterface.Out.SensorPositionFault,
                        oCyNo => #CyInterface.Out.CyNO,
                        ioManualGoWork := #CyInterface.Inout.ManualGoWork,
                        ioManualGoHome := #CyInterface.Inout.ManualGoHome,
                        ioAutoGoWork := #CyInterface.Inout.AutoGoWork,
                        ioAutoGoHome := #CyInterface.Inout.AutoGoHome,
                        ioGoWorkTime := #CyInterface.S.GoWorkTime,
                        ioGoHomeTime := #CyInterface.S.GoHomeTime,
                        ioWorkFaultTime := #CyInterface.S.WorkFaultTime,
                        ioHomeFaultTime := #CyInterface.S.HomeFaultTime,
                        ioBothSensorOnTime := #CyInterface.S.BothSensorOnTime,
                        ioPulse100mSP := #CyInterface.S.Pulse100mSP,
                        ioAutoGoWorkP := #CyInterface.S.AutoGoWorkP,
                        ioAutoGoHomeP := #CyInterface.S.AutoGoHomeP,
                        ioGoWork100mSP := #CyInterface.S.GoWork100mSP,
                        ioGoHome100mSP := #CyInterface.S.GoHome100mSP,
                        ioBothSensorOn100mSP := #CyInterface.S.BothSensorOn100mSP,
                        ioAlarm := #CyInterface.S.Alarm,
                        ioSpare1 := #CyInterface.S.spare1,
                        ioSpare2 := #CyInterface.S.spare2);
       //*******************************************************************************//
         POKE_BOOL(area := 16#84,
                   bitOffset := 4 * (#tpi MOD 2) + 0,
                   byteOffset :=  #tpi / 2,
                   dbNumber := #iDevAlarmDBNum,
                   value := #CyInterface.Out.GoWorkFault);
         POKE_BOOL(area := 16#84,
                   bitOffset := 4 * (#tpi MOD 2) + 1,
                   byteOffset :=  #tpi / 2,
                   dbNumber := #iDevAlarmDBNum,
                   value := #CyInterface.Out.GoHomeFault);
         POKE_BOOL(area := 16#84,
                   bitOffset := 4 * (#tpi MOD 2) + 2,
                   byteOffset :=  #tpi / 2,
                   dbNumber := #iDevAlarmDBNum,
                   value := #CyInterface.Out.SensorPositionFault);
       #CyInterface.Out.CyNO := INT_TO_BYTE(#tpi+1);
       //output
       #cyRSany.SyntaxID := 16#10;
       #cyRSany.DataType := 16#02;
       #cyRSany.RepetitionFactor := 16;
       #cyRSany.DB_Number := 0;
       #cyRSany.MemoryAreaAddress := 16#8700_0000 OR (SHL(IN := INT_TO_DWORD(6), N := 3));///
       //-----------------------------//
       #CyDSany.SyntaxID := 16#10;
       #CyDSany.DataType := 16#02;
       #CyDSany.RepetitionFactor := 16;
       #CyDSany.DB_Number := #iCyDBNO;
       #CyDSany.MemoryAreaAddress := 16#8400_0000 OR (SHL(IN := INT_TO_DWORD(#tpi* 22 + 6), N := 3));///
       #tpRetVal := BLKMOV(SRCBLK := #CyRany, DSTBLK => #CyDany);
       //******************************************************************************//


   END_FOR;
END_FUNCTION

FUNCTION "ST10Cyl_interface1-10" : Void   // FC1020, LAD
{ S7_Optimized_Access := 'FALSE' }
VERSION : 0.1
// stored: AutoNumber false, IsIECCheckEnabled false, SetENOAutomatically false, UDAEnableTagReadback false
   VAR_INPUT
      AlwaysON : Bool;
      E_stop : Bool;
   END_VAR
   VAR_TEMP
      tTest : Bool;
      i : Int;
   END_VAR
BEGIN

REGION Network 1 (SCL): Cylinder 1-10 IO Interface (SCL)
   IF "Station_Sys".Manual.Mode THEN

       FOR #i := 1 TO 100 BY 1

       DO
           "ST10Cylinder".Cy[#i].In.ManualOutputType := TRUE;

       END_FOR;

   END_IF;

   //Cylinder1 IO  A-Loading-01HorizontalCylinder
   //Input
   "ST10Cylinder".Cy[1].In.WorkPositionSensor := "iA-Loading-01HorizontalCylinderInWP";
   "ST10Cylinder".Cy[1].In.HomePositionSensor := "iA-Loading-01HorizontalCylinderInHP";
   //Output
   "oA-Loading-01HorizontalCylinderToWP" := "ST10Cylinder".Cy[1].Out.GoWorkPosition;
   "oA-Loading-01HorizontalCylinderToHP" := "ST10Cylinder".Cy[1].Out.GoHomePosition;

   //Cylinder2 IO  A-Loading-01UpDownTakeCylinder
   //Input
   "ST10Cylinder".Cy[2].In.WorkPositionSensor := "iA-Loading-01UpDownTakeCylinderInWP";
   "ST10Cylinder".Cy[2].In.HomePositionSensor := "iA-Loading-01UpDownTakeCylinderInHP";
   //Output
   "oA-Loading-01UpDownTakeCylinderToWP" := "ST10Cylinder".Cy[2].Out.GoWorkPosition;
   "oA-Loading-01UpDownTakeCylinderToHP" := "ST10Cylinder".Cy[2].Out.GoHomePosition;

   //Cylinder3 IO  A-Loading-02HorizontalCylinder
   //Input
   "ST10Cylinder".Cy[3].In.WorkPositionSensor := "iA-Loading-02HorizontalCylinderInWP"  ;
   "ST10Cylinder".Cy[3].In.HomePositionSensor := "iA-Loading-02HorizontalCylinderInHP"  ;
   //Output
   "oA-Loading-02HorizontalCylinderToWP" := "ST10Cylinder".Cy[3].Out.GoWorkPosition;
   "oA-Loading-02HorizontalCylinderToHP" := "ST10Cylinder".Cy[3].Out.GoHomePosition;

   //Cylinder4 IO     A-Loading-02UpDownTakeCylinder
   //Input
   "ST10Cylinder".Cy[4].In.WorkPositionSensor := "iA-Loading-02UpDownTakeCylinderInWP";
   "ST10Cylinder".Cy[4].In.HomePositionSensor := "iA-Loading-02UpDownTakeCylinderInHP";
   //Output
   "oA-Loading-02UpDownTakeCylinderToWP" := "ST10Cylinder".Cy[4].Out.GoWorkPosition;
   "oA-Loading-02UpDownTakeCylinderToHP" := "ST10Cylinder".Cy[4].Out.GoHomePosition;

   //Cylinder5 IO  B-PressFitting-01GripperCylinder
   //Input
   "ST10Cylinder".Cy[5].In.WorkPositionSensor := "iB-PressFitting-01GripperCylinderInWP";
   "ST10Cylinder".Cy[5].In.HomePositionSensor := "iB-PressFitting-01GripperCylinderInHP";
   //Output
   "oB-PressFitting-01GripperCylinderToWP" := "ST10Cylinder".Cy[5].Out.GoWorkPosition;
   "oB-PressFitting-01GripperCylinderToHP" := "ST10Cylinder".Cy[5].Out.GoHomePosition;

   //Cylinder6 IO  B-PressFitting-01Cylinder
   //Input
   "ST10Cylinder".Cy[6].In.WorkPositionSensor := "iB-PressFitting-01CylinderInWP" ;
   "ST10Cylinder".Cy[6].In.HomePositionSensor := "iB-PressFitting-01CylinderInHP" ;
   //Output
   "oB-PressFitting-01CylinderToWP" := "ST10Cylinder".Cy[6].Out.GoWorkPosition;
   "oB-PressFitting-01CylinderToHP" := "ST10Cylinder".Cy[6].Out.GoHomePosition;

   //Cylinder7 IO  B-PressFitting-02GripperCylinder
   //Input
   "ST10Cylinder".Cy[7].In.WorkPositionSensor := "iB-PressFitting-02GripperCylinderInWP";
   "ST10Cylinder".Cy[7].In.HomePositionSensor := "iB-PressFitting-02GripperCylinderInHP";
   //Output
   "oB-PressFitting-02GripperCylinderToWP" := "ST10Cylinder".Cy[7].Out.GoWorkPosition;
   "oB-PressFitting-02GripperCylinderToHP" := "ST10Cylinder".Cy[7].Out.GoHomePosition;

   //Cylinder8 IO  B-PressFitting-02Cylinder
   //Input
   "ST10Cylinder".Cy[8].In.WorkPositionSensor := "iB-PressFitting-02CylinderInWP";
   "ST10Cylinder".Cy[8].In.HomePositionSensor := "iB-PressFitting-02CylinderInHP";
   //Output
   "oB-PressFitting-02CylinderToWP" := "ST10Cylinder".Cy[8].Out.GoWorkPosition;
   "oB-PressFitting-02CylinderToHP" := "ST10Cylinder".Cy[8].Out.GoHomePosition;

   //Cylinder9 IO  C-LocationCylinder
   //Input
   "ST10Cylinder".Cy[9].In.WorkPositionSensor := "iC-LocationCylinderInWP";
   "ST10Cylinder".Cy[9].In.HomePositionSensor := "iC-LocationCylinderInHP";
   //Output
   "oC-LocationCylinderToWP" := "ST10Cylinder".Cy[9].Out.GoWorkPosition;
   "oC-LocationCylinderToHP" := "ST10Cylinder".Cy[9].Out.GoHomePosition;


   //Cylinder10 IO  Spare
   //Input
   "ST10Cylinder".Cy[10].In.WorkPositionSensor := "ST10Cylinder".Cy[10].Out.GoWorkPosition ;
   "ST10Cylinder".Cy[10].In.HomePositionSensor := "ST10Cylinder".Cy[10].Out.GoHomePosition ;
   //Output
   "ST10Cylinder".Cy[10].Out.GoWorkPosition := "ST10Cylinder".Cy[10].Out.GoWorkPosition;
   "ST10Cylinder".Cy[10].Out.GoHomePosition := "ST10Cylinder".Cy[10].Out.GoHomePosition;
END_REGION

REGION Network 2: CY1 interface A-Loading-01HorizontalCylinder
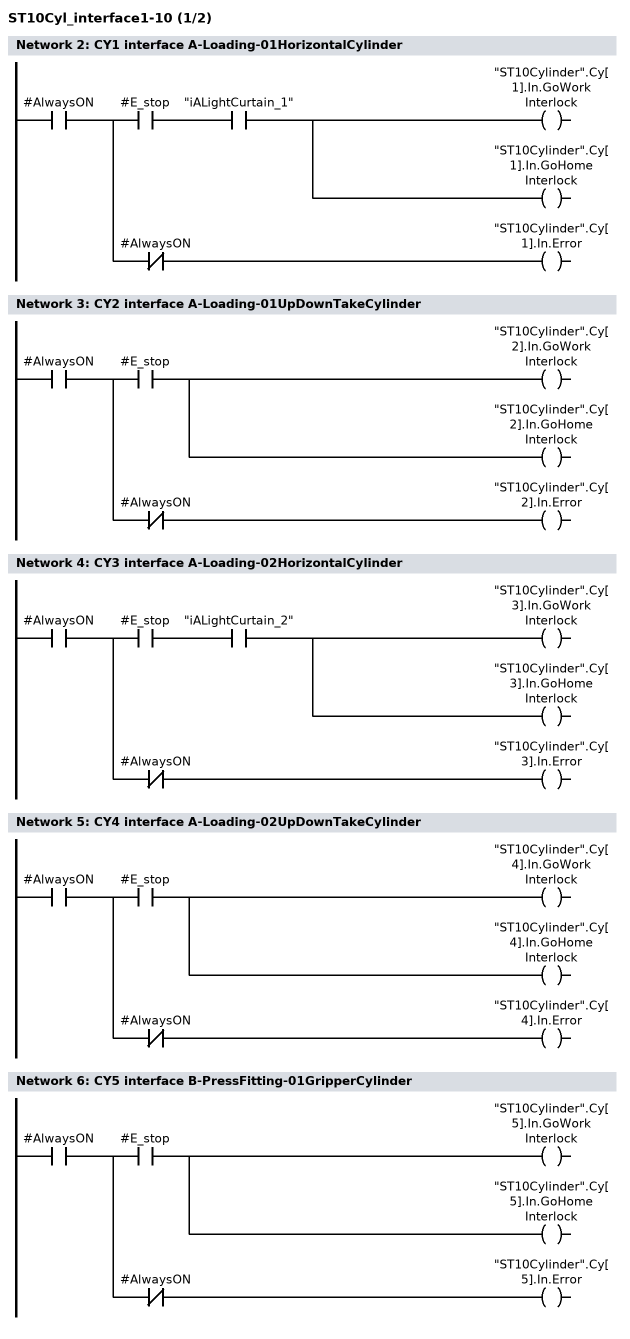
   RUNG wire#powerrail
      Contact( #AlwaysON )
      wire#w1
      Contact( #E_stop )
      Contact( "iALightCurtain_1" )
      wire#w2
      Coil( "ST10Cylinder".Cy[1].In.GoWorkInterlock )
   END_RUNG
   RUNG wire#w2
      Coil( "ST10Cylinder".Cy[1].In.GoHomeInterlock )
   END_RUNG
   RUNG wire#w1
      I_Contact( #AlwaysON )
      Coil( "ST10Cylinder".Cy[1].In.Error )
   END_RUNG
   // the same network as SCL:
   "ST10Cylinder".Cy[1].In.GoWorkInterlock := #AlwaysON AND #E_stop AND "iALightCurtain_1";
   "ST10Cylinder".Cy[1].In.GoHomeInterlock := #AlwaysON AND #E_stop AND "iALightCurtain_1";
   "ST10Cylinder".Cy[1].In.Error := #AlwaysON AND NOT #AlwaysON;
END_REGION

REGION Network 3: CY2 interface A-Loading-01UpDownTakeCylinder
   RUNG wire#powerrail
      Contact( #AlwaysON )
      wire#w1
      Contact( #E_stop )
      wire#w2
      Coil( "ST10Cylinder".Cy[2].In.GoWorkInterlock )
   END_RUNG
   RUNG wire#w2
      Coil( "ST10Cylinder".Cy[2].In.GoHomeInterlock )
   END_RUNG
   RUNG wire#w1
      I_Contact( #AlwaysON )
      Coil( "ST10Cylinder".Cy[2].In.Error )
   END_RUNG
   // the same network as SCL:
   "ST10Cylinder".Cy[2].In.GoWorkInterlock := #AlwaysON AND #E_stop;
   "ST10Cylinder".Cy[2].In.GoHomeInterlock := #AlwaysON AND #E_stop;
   "ST10Cylinder".Cy[2].In.Error := #AlwaysON AND NOT #AlwaysON;
END_REGION

REGION Network 4: CY3 interface A-Loading-02HorizontalCylinder
   RUNG wire#powerrail
      Contact( #AlwaysON )
      wire#w1
      Contact( #E_stop )
      Contact( "iALightCurtain_2" )
      wire#w2
      Coil( "ST10Cylinder".Cy[3].In.GoWorkInterlock )
   END_RUNG
   RUNG wire#w2
      Coil( "ST10Cylinder".Cy[3].In.GoHomeInterlock )
   END_RUNG
   RUNG wire#w1
      I_Contact( #AlwaysON )
      Coil( "ST10Cylinder".Cy[3].In.Error )
   END_RUNG
   // the same network as SCL:
   "ST10Cylinder".Cy[3].In.GoWorkInterlock := #AlwaysON AND #E_stop AND "iALightCurtain_2";
   "ST10Cylinder".Cy[3].In.GoHomeInterlock := #AlwaysON AND #E_stop AND "iALightCurtain_2";
   "ST10Cylinder".Cy[3].In.Error := #AlwaysON AND NOT #AlwaysON;
END_REGION

REGION Network 5: CY4 interface A-Loading-02UpDownTakeCylinder
   RUNG wire#powerrail
      Contact( #AlwaysON )
      wire#w1
      Contact( #E_stop )
      wire#w2
      Coil( "ST10Cylinder".Cy[4].In.GoWorkInterlock )
   END_RUNG
   RUNG wire#w2
      Coil( "ST10Cylinder".Cy[4].In.GoHomeInterlock )
   END_RUNG
   RUNG wire#w1
      I_Contact( #AlwaysON )
      Coil( "ST10Cylinder".Cy[4].In.Error )
   END_RUNG
   // the same network as SCL:
   "ST10Cylinder".Cy[4].In.GoWorkInterlock := #AlwaysON AND #E_stop;
   "ST10Cylinder".Cy[4].In.GoHomeInterlock := #AlwaysON AND #E_stop;
   "ST10Cylinder".Cy[4].In.Error := #AlwaysON AND NOT #AlwaysON;
END_REGION

REGION Network 6: CY5 interface B-PressFitting-01GripperCylinder
   RUNG wire#powerrail
      Contact( #AlwaysON )
      wire#w1
      Contact( #E_stop )
      wire#w2
      Coil( "ST10Cylinder".Cy[5].In.GoWorkInterlock )
   END_RUNG
   RUNG wire#w2
      Coil( "ST10Cylinder".Cy[5].In.GoHomeInterlock )
   END_RUNG
   RUNG wire#w1
      I_Contact( #AlwaysON )
      Coil( "ST10Cylinder".Cy[5].In.Error )
   END_RUNG
   // the same network as SCL:
   "ST10Cylinder".Cy[5].In.GoWorkInterlock := #AlwaysON AND #E_stop;
   "ST10Cylinder".Cy[5].In.GoHomeInterlock := #AlwaysON AND #E_stop;
   "ST10Cylinder".Cy[5].In.Error := #AlwaysON AND NOT #AlwaysON;
END_REGION

REGION Network 7: CY6 interface B-PressFitting-01Cylinder
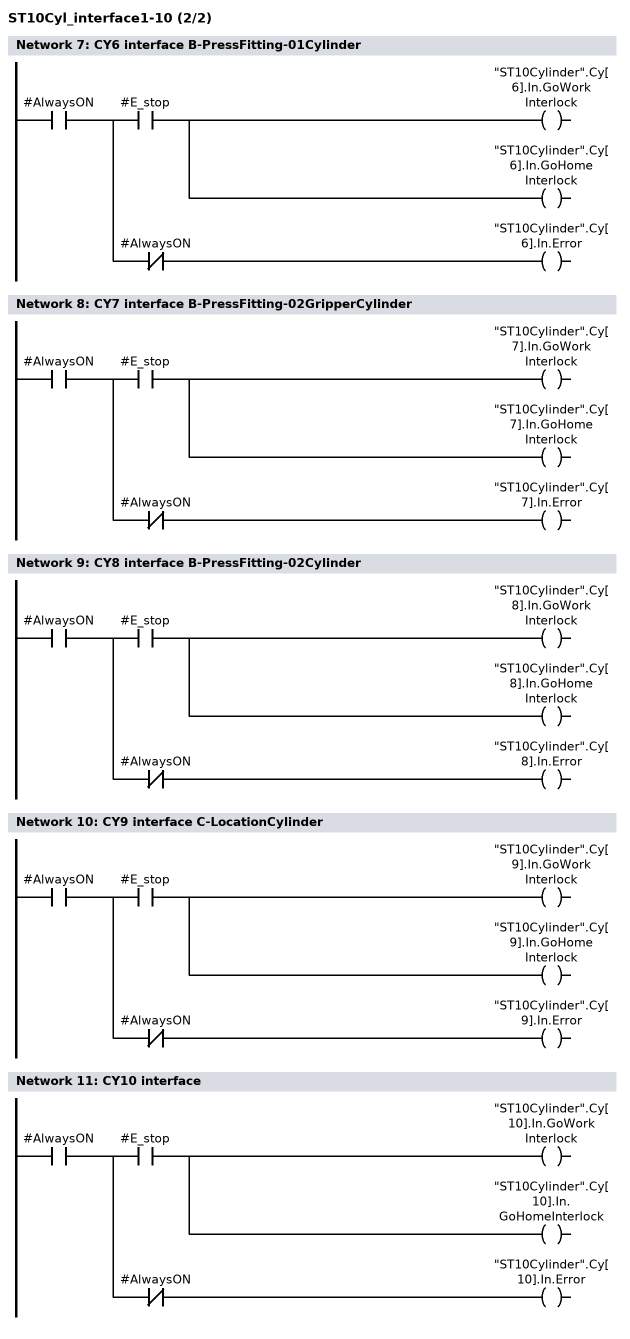
   RUNG wire#powerrail
      Contact( #AlwaysON )
      wire#w1
      Contact( #E_stop )
      wire#w2
      Coil( "ST10Cylinder".Cy[6].In.GoWorkInterlock )
   END_RUNG
   RUNG wire#w2
      Coil( "ST10Cylinder".Cy[6].In.GoHomeInterlock )
   END_RUNG
   RUNG wire#w1
      I_Contact( #AlwaysON )
      Coil( "ST10Cylinder".Cy[6].In.Error )
   END_RUNG
   // the same network as SCL:
   "ST10Cylinder".Cy[6].In.GoWorkInterlock := #AlwaysON AND #E_stop;
   "ST10Cylinder".Cy[6].In.GoHomeInterlock := #AlwaysON AND #E_stop;
   "ST10Cylinder".Cy[6].In.Error := #AlwaysON AND NOT #AlwaysON;
END_REGION

REGION Network 8: CY7 interface B-PressFitting-02GripperCylinder
   RUNG wire#powerrail
      Contact( #AlwaysON )
      wire#w1
      Contact( #E_stop )
      wire#w2
      Coil( "ST10Cylinder".Cy[7].In.GoWorkInterlock )
   END_RUNG
   RUNG wire#w2
      Coil( "ST10Cylinder".Cy[7].In.GoHomeInterlock )
   END_RUNG
   RUNG wire#w1
      I_Contact( #AlwaysON )
      Coil( "ST10Cylinder".Cy[7].In.Error )
   END_RUNG
   // the same network as SCL:
   "ST10Cylinder".Cy[7].In.GoWorkInterlock := #AlwaysON AND #E_stop;
   "ST10Cylinder".Cy[7].In.GoHomeInterlock := #AlwaysON AND #E_stop;
   "ST10Cylinder".Cy[7].In.Error := #AlwaysON AND NOT #AlwaysON;
END_REGION

REGION Network 9: CY8 interface B-PressFitting-02Cylinder
   RUNG wire#powerrail
      Contact( #AlwaysON )
      wire#w1
      Contact( #E_stop )
      wire#w2
      Coil( "ST10Cylinder".Cy[8].In.GoWorkInterlock )
   END_RUNG
   RUNG wire#w2
      Coil( "ST10Cylinder".Cy[8].In.GoHomeInterlock )
   END_RUNG
   RUNG wire#w1
      I_Contact( #AlwaysON )
      Coil( "ST10Cylinder".Cy[8].In.Error )
   END_RUNG
   // the same network as SCL:
   "ST10Cylinder".Cy[8].In.GoWorkInterlock := #AlwaysON AND #E_stop;
   "ST10Cylinder".Cy[8].In.GoHomeInterlock := #AlwaysON AND #E_stop;
   "ST10Cylinder".Cy[8].In.Error := #AlwaysON AND NOT #AlwaysON;
END_REGION

REGION Network 10: CY9 interface C-LocationCylinder
   RUNG wire#powerrail
      Contact( #AlwaysON )
      wire#w1
      Contact( #E_stop )
      wire#w2
      Coil( "ST10Cylinder".Cy[9].In.GoWorkInterlock )
   END_RUNG
   RUNG wire#w2
      Coil( "ST10Cylinder".Cy[9].In.GoHomeInterlock )
   END_RUNG
   RUNG wire#w1
      I_Contact( #AlwaysON )
      Coil( "ST10Cylinder".Cy[9].In.Error )
   END_RUNG
   // the same network as SCL:
   "ST10Cylinder".Cy[9].In.GoWorkInterlock := #AlwaysON AND #E_stop;
   "ST10Cylinder".Cy[9].In.GoHomeInterlock := #AlwaysON AND #E_stop;
   "ST10Cylinder".Cy[9].In.Error := #AlwaysON AND NOT #AlwaysON;
END_REGION

REGION Network 11: CY10 interface
   RUNG wire#powerrail
      Contact( #AlwaysON )
      wire#w1
      Contact( #E_stop )
      wire#w2
      Coil( "ST10Cylinder".Cy[10].In.GoWorkInterlock )
   END_RUNG
   RUNG wire#w2
      Coil( "ST10Cylinder".Cy[10].In.GoHomeInterlock )
   END_RUNG
   RUNG wire#w1
      I_Contact( #AlwaysON )
      Coil( "ST10Cylinder".Cy[10].In.Error )
   END_RUNG
   // the same network as SCL:
   "ST10Cylinder".Cy[10].In.GoWorkInterlock := #AlwaysON AND #E_stop;
   "ST10Cylinder".Cy[10].In.GoHomeInterlock := #AlwaysON AND #E_stop;
   "ST10Cylinder".Cy[10].In.Error := #AlwaysON AND NOT #AlwaysON;
END_REGION
END_FUNCTION

FUNCTION "ST10Cyl_interface11-20" : Void   // FC1021, LAD
{ S7_Optimized_Access := 'FALSE' }
// stored: AutoNumber false, SetENOAutomatically false
   VAR_INPUT
      AlwaysON : Bool;
      E_stop : Bool;
   END_VAR
   VAR_TEMP
      tTest : Bool;
   END_VAR
BEGIN

REGION Network 1 (SCL): Cylinder 11-20 IO Interface (SCL)

   //Cylinder11 IO   E-NG-01NGLocationCylinder
   //Input
   "ST10Cylinder".Cy[11].In.WorkPositionSensor := "iE-NG-01NGLocationCylinderInWP";
   "ST10Cylinder".Cy[11].In.HomePositionSensor := "iE-NG-01NGLocationCylinderInHP";
   //Output
   //"oE-NG-01NGLocationCylinderToWP" := "ST10Cylinder".Cy[11].Out.GoWorkPosition;
   //"oE-NG-01NGLocationCylinderToHP" := "ST10Cylinder".Cy[11].Out.GoHomePosition;

   //Cylinder12 IO  E-NG-02NGLocationCylinder
   //Input
   "ST10Cylinder".Cy[12].In.WorkPositionSensor := "iE-NG-02NGLocationCylinderInWP";
   "ST10Cylinder".Cy[12].In.HomePositionSensor := "iE-NG-02NGLocationCylinderInHP";
   //Output
   //"oE-NG-02NGLocationCylinderToWP" := "ST10Cylinder".Cy[12].Out.GoWorkPosition;
   //"oE-NG-02NGLocationCylinderToHP" := "ST10Cylinder".Cy[12].Out.GoHomePosition;

   //Cylinder13 IO  F-ROOBT1Gripper1Cylinder
   //Input
   "KukaRobot1_CtrlDB".sPLCtoROB.User.Gripper.DI129_Grip1WP:="ST10Cylinder".Cy[13].In.WorkPositionSensor := "iF-ROOBT1Gripper1CylinderInWP" ;
   "KukaRobot1_CtrlDB".sPLCtoROB.User.Gripper.DI130_Grip1HP := "ST10Cylinder".Cy[13].In.HomePositionSensor := "iF-ROOBT1Gripper1CylinderInHP" ;//"TON".TON[0].Q;

   IF  NOT "Robot_DB".Control.Robot1GripControl THEN
       //Output
       "oF-ROOBT1Gripper1CylinderToWP" := "KukaRobot1_CtrlDB".sROBtoPLC.User.Gripper.DO129_Grip1GoWork;
       "oF-ROOBT1Gripper1CylinderToHP" := "KukaRobot1_CtrlDB".sROBtoPLC.User.Gripper.DO130_Grip1GoHome;
   ELSE
       //Output
       "oF-ROOBT1Gripper1CylinderToWP" := "ST10Cylinder".Cy[13].Out.GoWorkPosition;
       "oF-ROOBT1Gripper1CylinderToHP" := "ST10Cylinder".Cy[13].Out.GoHomePosition;
   END_IF;
   "TON".TON[0](IN:="oF-ROOBT1Gripper1CylinderToHP" AND NOT"iF-ROOBT1Gripper1CylinderInWP",PT:=T#500MS);


   //Cylinder14 IO  F-ROOBT1Gripper2Cylinder
   //Input
   "KukaRobot1_CtrlDB".sPLCtoROB.User.Gripper.DI131_Grip2WP:="ST10Cylinder".Cy[14].In.WorkPositionSensor := "iF-ROOBT1Gripper2CylinderInWP";
   "KukaRobot1_CtrlDB".sPLCtoROB.User.Gripper.DI132_Grip2HP:="ST10Cylinder".Cy[14].In.HomePositionSensor := "iF-ROOBT1Gripper2CylinderInHP";

   IF NOT "Robot_DB".Control.Robot1GripControl THEN
       //Output
       "oF-ROOBT1Gripper2CylinderToWP" :="ST10Cylinder".Cy[14].Inout.AutoGoWork:="KukaRobot1_CtrlDB".sROBtoPLC.User.Gripper.DO131_Grip2GoWork;
       "oF-ROOBT1Gripper2CylinderToHP" :="ST10Cylinder".Cy[14].Inout.AutoGoHome:="KukaRobot1_CtrlDB".sROBtoPLC.User.Gripper.DO132_Grip2GoHome;
   ELSE
       //Output
       "oF-ROOBT1Gripper2CylinderToWP" := "ST10Cylinder".Cy[14].Out.GoWorkPosition;
       "oF-ROOBT1Gripper2CylinderToHP" := "ST10Cylinder".Cy[14].Out.GoHomePosition;
   END_IF;


   //Cylinder15 IO  F-ROOBT2Gripper1Cylinder
   //Input
   "KukaRobot2_CtrlDB".sPLCtoROB.User.Gripper.DI129_Grip1WP:="ST10Cylinder".Cy[15].In.WorkPositionSensor := "iF-ROOBT2Gripper1CylinderInWP";
   "KukaRobot2_CtrlDB".sPLCtoROB.User.Gripper.DI130_Grip1HP := "ST10Cylinder".Cy[15].In.HomePositionSensor :="iF-ROOBT2Gripper1CylinderInHP";

   IF NOT "Robot_DB".Control.Robot2GripControl THEN
       //Output
       "oF-ROOBT2Gripper1CylinderToWP" :="ST10Cylinder".Cy[15].Inout.AutoGoWork:="KukaRobot2_CtrlDB".sROBtoPLC.User.Gripper.DO129_Grip1GoWork;
       "oF-ROOBT2Gripper1CylinderToHP" :="ST10Cylinder".Cy[15].Inout.AutoGoHome:="KukaRobot2_CtrlDB".sROBtoPLC.User.Gripper.DO130_Grip1GoHome;
   ELSE
       //Output
       "oF-ROOBT2Gripper1CylinderToWP" := "ST10Cylinder".Cy[15].Out.GoWorkPosition;
       "oF-ROOBT2Gripper1CylinderToHP" := "ST10Cylinder".Cy[15].Out.GoHomePosition;
   END_IF;



   //Cylinder16 IO  F-ROOBT2Gripper2Cylinder
   //Input
   "KukaRobot2_CtrlDB".sPLCtoROB.User.Gripper.DI131_Grip2WP:="ST10Cylinder".Cy[16].In.WorkPositionSensor := "iF-ROOBT2Gripper2CylinderInWP";
   "KukaRobot2_CtrlDB".sPLCtoROB.User.Gripper.DI132_Grip2HP:="ST10Cylinder".Cy[16].In.HomePositionSensor := "iF-ROOBT2Gripper2CylinderInHP";

   IF NOT "Robot_DB".Control.Robot2GripControl THEN
       //Output
       "oF-ROOBT2Gripper2CylinderToWP" :="ST10Cylinder".Cy[16].Inout.AutoGoWork:= "KukaRobot2_CtrlDB".sROBtoPLC.User.Gripper.DO131_Grip2GoWork;
       "oF-ROOBT2Gripper2CylinderToHP" :="ST10Cylinder".Cy[16].Inout.AutoGoHome:= "KukaRobot2_CtrlDB".sROBtoPLC.User.Gripper.DO132_Grip2GoHome;
   ELSE
       //Output
       "oF-ROOBT2Gripper2CylinderToWP" := "ST10Cylinder".Cy[16].Out.GoWorkPosition;
       "oF-ROOBT2Gripper2CylinderToHP" := "ST10Cylinder".Cy[16].Out.GoHomePosition;
   END_IF;

   //Cylinder17 IO  F-ROOBT3Gripper1Cylinder
   //Input
   "KukaRobot3_CtrlDB".sPLCtoROB.User.Gripper.DI129_Grip1WP:="ST10Cylinder".Cy[17].In.WorkPositionSensor := "iF-ROOBT3Gripper1CylinderInWP";
   "KukaRobot3_CtrlDB".sPLCtoROB.User.Gripper.DI130_Grip1HP:="ST10Cylinder".Cy[17].In.HomePositionSensor := "iF-ROOBT3Gripper1CylinderInHP";

   IF NOT "Robot_DB".Control.Robot3GripControl THEN
       //Output
       "oF-ROOBT3Gripper1CylinderToWP" :="ST10Cylinder".Cy[17].Inout.AutoGoWork:="KukaRobot3_CtrlDB".sROBtoPLC.User.Gripper.DO129_Grip1GoWork;
       "oF-ROOBT3Gripper1CylinderToHP" :="ST10Cylinder".Cy[17].Inout.AutoGoHome:="KukaRobot3_CtrlDB".sROBtoPLC.User.Gripper.DO130_Grip1GoHome;
   ELSE
       //Output
       "oF-ROOBT3Gripper1CylinderToWP" := "ST10Cylinder".Cy[17].Out.GoWorkPosition;
       "oF-ROOBT3Gripper1CylinderToHP" := "ST10Cylinder".Cy[17].Out.GoHomePosition;
   END_IF;


   //Cylinder18 IO  F-ROOBT3Gripper2Cylinder
   //Input
   "KukaRobot3_CtrlDB".sPLCtoROB.User.Gripper.DI131_Grip2WP:="ST10Cylinder".Cy[18].In.WorkPositionSensor := "iF-ROOBT3Gripper2CylinderInWP";
   "KukaRobot3_CtrlDB".sPLCtoROB.User.Gripper.DI132_Grip2HP := "ST10Cylinder".Cy[18].In.HomePositionSensor := "iF-ROOBT3Gripper2CylinderInHP";//"TON".TON[1].Q;

   IF NOT "Robot_DB".Control.Robot3GripControl THEN
       //Output
       "oF-ROOBT3Gripper2CylinderToWP" :="ST10Cylinder".Cy[18].Inout.AutoGoWork:="KukaRobot3_CtrlDB".sROBtoPLC.User.Gripper.DO131_Grip2GoWork;
       "oF-ROOBT3Gripper2CylinderToHP" :="ST10Cylinder".Cy[18].Inout.AutoGoHome:="KukaRobot3_CtrlDB".sROBtoPLC.User.Gripper.DO132_Grip2GoHome;
   ELSE
       //Output
       "oF-ROOBT3Gripper2CylinderToWP" := "ST10Cylinder".Cy[18].Out.GoWorkPosition;
       "oF-ROOBT3Gripper2CylinderToHP" := "ST10Cylinder".Cy[18].Out.GoHomePosition;
   END_IF;

   "TON".TON[1](IN := "oF-ROOBT3Gripper2CylinderToHP" AND NOT "iF-ROOBT3Gripper2CylinderInWP",
                PT := T#500MS);

   (*
   //Cylinder19 IO  D-washer Loading Horizontal
   //Input
   "ST10Cylinder".Cy[19].In.WorkPositionSensor := ("D-washer Loading Cylinder Middle Cylinder InHP" AND "D-washer Loading Horizontal Cylinder InWP")
                                               OR ("D-washer Loading Cylinder Middle Cylinder InWP" AND "D-washer Loading Horizontal Cylinder InWP1");
   "ST10Cylinder".Cy[19].In.HomePositionSensor := "D-washer Loading Horizontal Cylinder InHP";
   //Output
   "D-washer Loading Horizontal Cylinder ToWP" := "ST10Cylinder".Cy[19].Out.GoWorkPosition;
   "D-washer Loading Horizontal Cylinder ToHP" := "ST10Cylinder".Cy[19].Out.GoHomePosition;

   //Cylinder20 IO  D-washer Loading Cylinder Middle
   //Input
   "ST10Cylinder".Cy[20].In.WorkPositionSensor := "D-washer Loading Cylinder Middle Cylinder InWP";
   "ST10Cylinder".Cy[20].In.HomePositionSensor := "D-washer Loading Cylinder Middle Cylinder InHP";
   //Output
   "D-washer Loading Cylinder Middle Cylinder ToWP" := "ST10Cylinder".Cy[20].Out.GoWorkPosition;
   "D-washer Loading Cylinder Middle Cylinder ToHP" := "ST10Cylinder".Cy[20].Out.GoHomePosition;
   *)
END_REGION

REGION Network 2: CY11 interface E-NG-01NGLocationCylinder
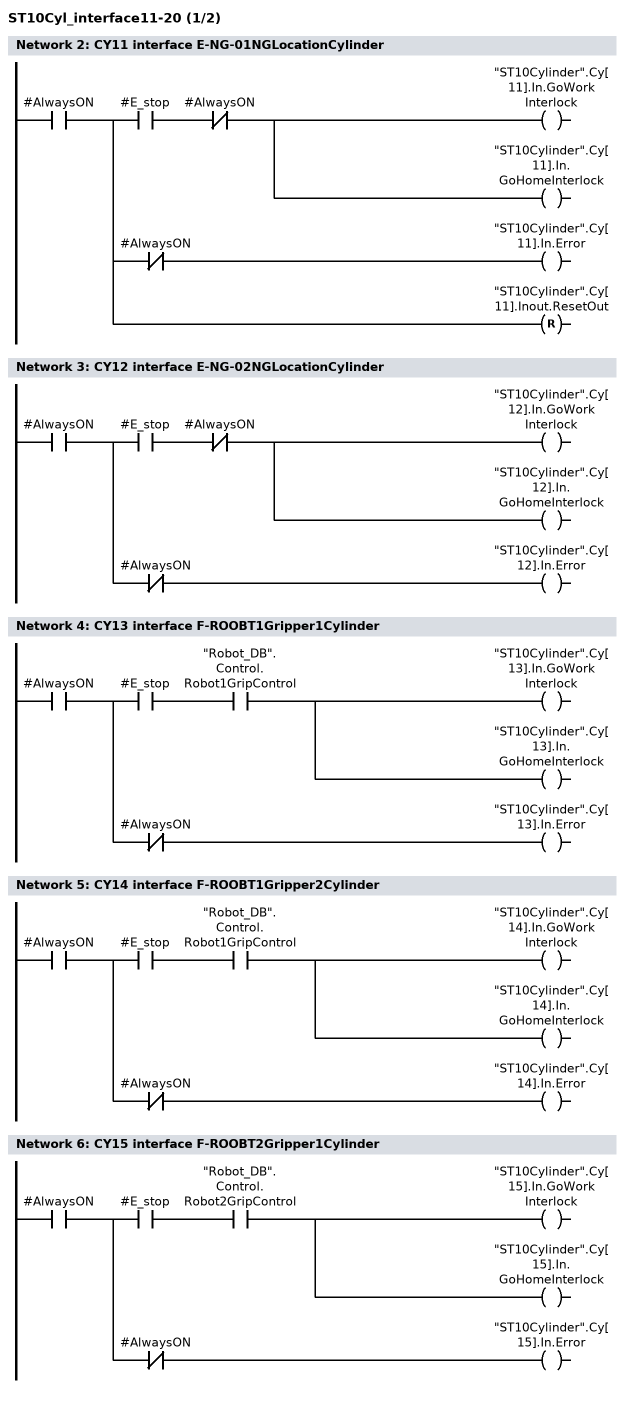
   RUNG wire#powerrail
      Contact( #AlwaysON )
      wire#w1
      Contact( #E_stop )
      I_Contact( #AlwaysON )
      wire#w2
      Coil( "ST10Cylinder".Cy[11].In.GoWorkInterlock )
   END_RUNG
   RUNG wire#w2
      Coil( "ST10Cylinder".Cy[11].In.GoHomeInterlock )
   END_RUNG
   RUNG wire#w1
      I_Contact( #AlwaysON )
      Coil( "ST10Cylinder".Cy[11].In.Error )
   END_RUNG
   RUNG wire#w1
      R_Coil( "ST10Cylinder".Cy[11].Inout.ResetOut )
   END_RUNG
   // the same network as SCL:
   "ST10Cylinder".Cy[11].In.GoWorkInterlock := #AlwaysON AND #E_stop AND NOT #AlwaysON;
   "ST10Cylinder".Cy[11].In.GoHomeInterlock := #AlwaysON AND #E_stop AND NOT #AlwaysON;
   "ST10Cylinder".Cy[11].In.Error := #AlwaysON AND NOT #AlwaysON;
   IF #AlwaysON THEN "ST10Cylinder".Cy[11].Inout.ResetOut := FALSE; END_IF;
END_REGION

REGION Network 3: CY12 interface E-NG-02NGLocationCylinder
   RUNG wire#powerrail
      Contact( #AlwaysON )
      wire#w1
      Contact( #E_stop )
      I_Contact( #AlwaysON )
      wire#w2
      Coil( "ST10Cylinder".Cy[12].In.GoWorkInterlock )
   END_RUNG
   RUNG wire#w2
      Coil( "ST10Cylinder".Cy[12].In.GoHomeInterlock )
   END_RUNG
   RUNG wire#w1
      I_Contact( #AlwaysON )
      Coil( "ST10Cylinder".Cy[12].In.Error )
   END_RUNG
   // the same network as SCL:
   "ST10Cylinder".Cy[12].In.GoWorkInterlock := #AlwaysON AND #E_stop AND NOT #AlwaysON;
   "ST10Cylinder".Cy[12].In.GoHomeInterlock := #AlwaysON AND #E_stop AND NOT #AlwaysON;
   "ST10Cylinder".Cy[12].In.Error := #AlwaysON AND NOT #AlwaysON;
END_REGION

REGION Network 4: CY13 interface F-ROOBT1Gripper1Cylinder
   RUNG wire#powerrail
      Contact( #AlwaysON )
      wire#w1
      Contact( #E_stop )
      Contact( "Robot_DB".Control.Robot1GripControl )
      wire#w2
      Coil( "ST10Cylinder".Cy[13].In.GoWorkInterlock )
   END_RUNG
   RUNG wire#w2
      Coil( "ST10Cylinder".Cy[13].In.GoHomeInterlock )
   END_RUNG
   RUNG wire#w1
      I_Contact( #AlwaysON )
      Coil( "ST10Cylinder".Cy[13].In.Error )
   END_RUNG
   // the same network as SCL:
   "ST10Cylinder".Cy[13].In.GoWorkInterlock := #AlwaysON AND #E_stop AND "Robot_DB".Control.Robot1GripControl;
   "ST10Cylinder".Cy[13].In.GoHomeInterlock := #AlwaysON AND #E_stop AND "Robot_DB".Control.Robot1GripControl;
   "ST10Cylinder".Cy[13].In.Error := #AlwaysON AND NOT #AlwaysON;
END_REGION

REGION Network 5: CY14 interface F-ROOBT1Gripper2Cylinder
   RUNG wire#powerrail
      Contact( #AlwaysON )
      wire#w1
      Contact( #E_stop )
      Contact( "Robot_DB".Control.Robot1GripControl )
      wire#w2
      Coil( "ST10Cylinder".Cy[14].In.GoWorkInterlock )
   END_RUNG
   RUNG wire#w2
      Coil( "ST10Cylinder".Cy[14].In.GoHomeInterlock )
   END_RUNG
   RUNG wire#w1
      I_Contact( #AlwaysON )
      Coil( "ST10Cylinder".Cy[14].In.Error )
   END_RUNG
   // the same network as SCL:
   "ST10Cylinder".Cy[14].In.GoWorkInterlock := #AlwaysON AND #E_stop AND "Robot_DB".Control.Robot1GripControl;
   "ST10Cylinder".Cy[14].In.GoHomeInterlock := #AlwaysON AND #E_stop AND "Robot_DB".Control.Robot1GripControl;
   "ST10Cylinder".Cy[14].In.Error := #AlwaysON AND NOT #AlwaysON;
END_REGION

REGION Network 6: CY15 interface F-ROOBT2Gripper1Cylinder
   RUNG wire#powerrail
      Contact( #AlwaysON )
      wire#w1
      Contact( #E_stop )
      Contact( "Robot_DB".Control.Robot2GripControl )
      wire#w2
      Coil( "ST10Cylinder".Cy[15].In.GoWorkInterlock )
   END_RUNG
   RUNG wire#w2
      Coil( "ST10Cylinder".Cy[15].In.GoHomeInterlock )
   END_RUNG
   RUNG wire#w1
      I_Contact( #AlwaysON )
      Coil( "ST10Cylinder".Cy[15].In.Error )
   END_RUNG
   // the same network as SCL:
   "ST10Cylinder".Cy[15].In.GoWorkInterlock := #AlwaysON AND #E_stop AND "Robot_DB".Control.Robot2GripControl;
   "ST10Cylinder".Cy[15].In.GoHomeInterlock := #AlwaysON AND #E_stop AND "Robot_DB".Control.Robot2GripControl;
   "ST10Cylinder".Cy[15].In.Error := #AlwaysON AND NOT #AlwaysON;
END_REGION

REGION Network 7: CY16 interface F-ROOBT2Gripper2Cylinder
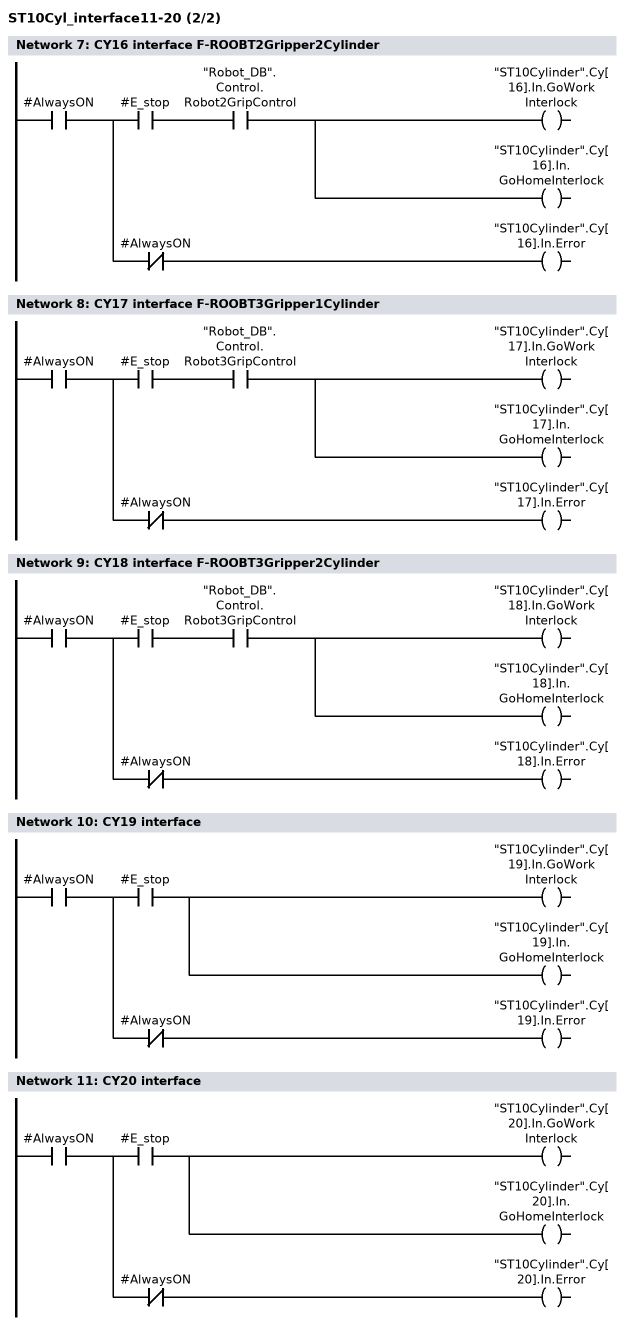
   RUNG wire#powerrail
      Contact( #AlwaysON )
      wire#w1
      Contact( #E_stop )
      Contact( "Robot_DB".Control.Robot2GripControl )
      wire#w2
      Coil( "ST10Cylinder".Cy[16].In.GoWorkInterlock )
   END_RUNG
   RUNG wire#w2
      Coil( "ST10Cylinder".Cy[16].In.GoHomeInterlock )
   END_RUNG
   RUNG wire#w1
      I_Contact( #AlwaysON )
      Coil( "ST10Cylinder".Cy[16].In.Error )
   END_RUNG
   // the same network as SCL:
   "ST10Cylinder".Cy[16].In.GoWorkInterlock := #AlwaysON AND #E_stop AND "Robot_DB".Control.Robot2GripControl;
   "ST10Cylinder".Cy[16].In.GoHomeInterlock := #AlwaysON AND #E_stop AND "Robot_DB".Control.Robot2GripControl;
   "ST10Cylinder".Cy[16].In.Error := #AlwaysON AND NOT #AlwaysON;
END_REGION

REGION Network 8: CY17 interface F-ROOBT3Gripper1Cylinder
   RUNG wire#powerrail
      Contact( #AlwaysON )
      wire#w1
      Contact( #E_stop )
      Contact( "Robot_DB".Control.Robot3GripControl )
      wire#w2
      Coil( "ST10Cylinder".Cy[17].In.GoWorkInterlock )
   END_RUNG
   RUNG wire#w2
      Coil( "ST10Cylinder".Cy[17].In.GoHomeInterlock )
   END_RUNG
   RUNG wire#w1
      I_Contact( #AlwaysON )
      Coil( "ST10Cylinder".Cy[17].In.Error )
   END_RUNG
   // the same network as SCL:
   "ST10Cylinder".Cy[17].In.GoWorkInterlock := #AlwaysON AND #E_stop AND "Robot_DB".Control.Robot3GripControl;
   "ST10Cylinder".Cy[17].In.GoHomeInterlock := #AlwaysON AND #E_stop AND "Robot_DB".Control.Robot3GripControl;
   "ST10Cylinder".Cy[17].In.Error := #AlwaysON AND NOT #AlwaysON;
END_REGION

REGION Network 9: CY18 interface F-ROOBT3Gripper2Cylinder
   RUNG wire#powerrail
      Contact( #AlwaysON )
      wire#w1
      Contact( #E_stop )
      Contact( "Robot_DB".Control.Robot3GripControl )
      wire#w2
      Coil( "ST10Cylinder".Cy[18].In.GoWorkInterlock )
   END_RUNG
   RUNG wire#w2
      Coil( "ST10Cylinder".Cy[18].In.GoHomeInterlock )
   END_RUNG
   RUNG wire#w1
      I_Contact( #AlwaysON )
      Coil( "ST10Cylinder".Cy[18].In.Error )
   END_RUNG
   // the same network as SCL:
   "ST10Cylinder".Cy[18].In.GoWorkInterlock := #AlwaysON AND #E_stop AND "Robot_DB".Control.Robot3GripControl;
   "ST10Cylinder".Cy[18].In.GoHomeInterlock := #AlwaysON AND #E_stop AND "Robot_DB".Control.Robot3GripControl;
   "ST10Cylinder".Cy[18].In.Error := #AlwaysON AND NOT #AlwaysON;
END_REGION

REGION Network 10: CY19 interface
   RUNG wire#powerrail
      Contact( #AlwaysON )
      wire#w1
      Contact( #E_stop )
      wire#w2
      Coil( "ST10Cylinder".Cy[19].In.GoWorkInterlock )
   END_RUNG
   RUNG wire#w2
      Coil( "ST10Cylinder".Cy[19].In.GoHomeInterlock )
   END_RUNG
   RUNG wire#w1
      I_Contact( #AlwaysON )
      Coil( "ST10Cylinder".Cy[19].In.Error )
   END_RUNG
   // the same network as SCL:
   "ST10Cylinder".Cy[19].In.GoWorkInterlock := #AlwaysON AND #E_stop;
   "ST10Cylinder".Cy[19].In.GoHomeInterlock := #AlwaysON AND #E_stop;
   "ST10Cylinder".Cy[19].In.Error := #AlwaysON AND NOT #AlwaysON;
END_REGION

REGION Network 11: CY20 interface
   RUNG wire#powerrail
      Contact( #AlwaysON )
      wire#w1
      Contact( #E_stop )
      wire#w2
      Coil( "ST10Cylinder".Cy[20].In.GoWorkInterlock )
   END_RUNG
   RUNG wire#w2
      Coil( "ST10Cylinder".Cy[20].In.GoHomeInterlock )
   END_RUNG
   RUNG wire#w1
      I_Contact( #AlwaysON )
      Coil( "ST10Cylinder".Cy[20].In.Error )
   END_RUNG
   // the same network as SCL:
   "ST10Cylinder".Cy[20].In.GoWorkInterlock := #AlwaysON AND #E_stop;
   "ST10Cylinder".Cy[20].In.GoHomeInterlock := #AlwaysON AND #E_stop;
   "ST10Cylinder".Cy[20].In.Error := #AlwaysON AND NOT #AlwaysON;
END_REGION
END_FUNCTION

FUNCTION "ST10Cyl_interface21-30" : Void   // FC1022, LAD
{ S7_Optimized_Access := 'FALSE' }
// stored: AutoNumber false, SetENOAutomatically false
   VAR_INPUT
      AlwaysON : Bool;
      E_stop : Bool;
   END_VAR
   VAR_TEMP
      tTest : Bool;
   END_VAR
BEGIN

REGION Network 1 (SCL): Cylinder 21-30 IO Interface (SCL)

   //Cylinder21 IO  H-shaftLiftingLiftingCylinder
   //Input
   "ST10Cylinder".Cy[21].In.WorkPositionSensor := "iH-shaftLiftingLiftingCylinderInWP" ;
   "ST10Cylinder".Cy[21].In.HomePositionSensor := "iH-shaftLiftingLiftingCylinderInHP" ;
   //Output
   "oH-shaftLiftingLiftingCylinderToWP" := "ST10Cylinder".Cy[21].Out.GoWorkPosition;
   "oH-shaftLiftingLiftingCylinderToHP" := "ST10Cylinder".Cy[21].Out.GoHomePosition;

   //Cylinder22 IO  H-shaftLiftingPalletLocationCylinder
   //Input
   "ST10Cylinder".Cy[22].In.WorkPositionSensor := "iH-shaftLiftingPalletLocationCylinderInWP" ;
   "ST10Cylinder".Cy[22].In.HomePositionSensor :="iH-shaftLiftingPalletLocationCylinderInHP"  ;
   //Output
   "oH-shaftLiftingPalletLocationCylinderToWP" := "ST10Cylinder".Cy[22].Out.GoWorkPosition;
   "oH-shaftLiftingPalletLocationCylinderToHP" := "ST10Cylinder".Cy[22].Out.GoHomePosition;

   //Cylinder23 IO  H-shaftLoadingStopperCylinder1
   //Input
   "ST10Cylinder".Cy[23].In.WorkPositionSensor := "oH-shaftLoadingStopperCylinder1_ToWP";
   "ST10Cylinder".Cy[23].In.HomePositionSensor := "oH-shaftLoadingStopperCylinder1_ToHP" ;
   //Output
   "oH-shaftLoadingStopperCylinder1_ToWP" := "ST10Cylinder".Cy[23].Out.GoWorkPosition;
   "oH-shaftLoadingStopperCylinder1_ToHP" := "ST10Cylinder".Cy[23].Out.GoHomePosition;

   //Cylinder24 IO  H-shaftLoadingStopperCylinder2
   //Input
   "ST10Cylinder".Cy[24].In.WorkPositionSensor := "oH-shaftLoadingStopperCylinder2_ToWP" ;
   "ST10Cylinder".Cy[24].In.HomePositionSensor := "oH-shaftLoadingStopperCylinder2_ToHP";
   //Output
   "oH-shaftLoadingStopperCylinder2_ToWP" := "ST10Cylinder".Cy[24].Out.GoWorkPosition;
   "oH-shaftLoadingStopperCylinder2_ToHP" := "ST10Cylinder".Cy[24].Out.GoHomePosition;

   //Cylinder25 IO  H-shaftLoadingStopperCylinder3
   //Input
   "ST10Cylinder".Cy[25].In.WorkPositionSensor := "oH-shaftLoadingStopperCylinder3_ToWP";
   "ST10Cylinder".Cy[25].In.HomePositionSensor := "oH-shaftLoadingStopperCylinder3_ToHP";
   //Output
   "oH-shaftLoadingStopperCylinder3_ToWP" := "ST10Cylinder".Cy[25].Out.GoWorkPosition;
   "oH-shaftLoadingStopperCylinder3_ToHP" := "ST10Cylinder".Cy[25].Out.GoHomePosition;

   //Cylinder26 H-shaftLoadingStopperCylinder4
   //Input
   "ST10Cylinder".Cy[26].In.WorkPositionSensor := "oH-shaftLoadingStopperCylinder4_ToWP";
   "ST10Cylinder".Cy[26].In.HomePositionSensor := "oH-shaftLoadingStopperCylinder4_ToHP" ;
   //Output
   "oH-shaftLoadingStopperCylinder4_ToWP" := "ST10Cylinder".Cy[26].Out.GoWorkPosition;
   "oH-shaftLoadingStopperCylinder4_ToHP" := "ST10Cylinder".Cy[26].Out.GoHomePosition;

   //Cylinder27 H-shaftTakeStopperCylinder1
   //Input
   "ST10Cylinder".Cy[27].In.WorkPositionSensor :="oH-shaftTakeStopperCylinder1_ToWP" ;
   "ST10Cylinder".Cy[27].In.HomePositionSensor :="oH-shaftTakeStopperCylinder1_ToHP";
   //Output
   "oH-shaftTakeStopperCylinder1_ToWP" :="ST10Cylinder".Cy[27].Out.GoWorkPosition;
   "oH-shaftTakeStopperCylinder1_ToHP" := "ST10Cylinder".Cy[27].Out.GoHomePosition;

   //Cylinder28 H-shaftTakeStopperCylinder2
   //Input
   "ST10Cylinder".Cy[28].In.WorkPositionSensor :="oH-shaftTakeStopperCylinder2_ToWP" ;
   "ST10Cylinder".Cy[28].In.HomePositionSensor := "oH-shaftTakeStopperCylinder2_ToHP";
   //Output
   "oH-shaftTakeStopperCylinder2_ToWP" := "ST10Cylinder".Cy[28].Out.GoWorkPosition;
   "oH-shaftTakeStopperCylinder2_ToHP" := "ST10Cylinder".Cy[28].Out.GoHomePosition;

   //Cylinder29 H-shaftTakeStopperCylinder3
   //Input
   "ST10Cylinder".Cy[29].In.WorkPositionSensor :="oH-shaftTakeStopperCylinder3_ToWP" ;
   "ST10Cylinder".Cy[29].In.HomePositionSensor :="oH-shaftTakeStopperCylinder3_ToHP";
   //Output
   "oH-shaftTakeStopperCylinder3_ToWP" := "ST10Cylinder".Cy[29].Out.GoWorkPosition;
   "oH-shaftTakeStopperCylinder3_ToHP" := "ST10Cylinder".Cy[29].Out.GoHomePosition;

    (*
    //Cylinder30 H-shaftLoadingStopperCylinder4_2  
   // //Input
   "ST10Cylinder".Cy[30].In.WorkPositionSensor := "oH-shaftLoadingStopperCylinder4_2";
   "ST10Cylinder".Cy[30].In.HomePositionSensor := NOT "oH-shaftLoadingStopperCylinder4_2";
   // //Output
    "oH-shaftLoadingStopperCylinder4_2" := "ST10Cylinder".Cy[30].Out.GoWorkPosition;
    "Feeding washer  lift Cylinder ToHP" := "ST10Cylinder".Cy[30].Out.GoHomePosition;
   *)
END_REGION

REGION Network 2: CY21 interface H-shaftLiftingLiftingCylinder
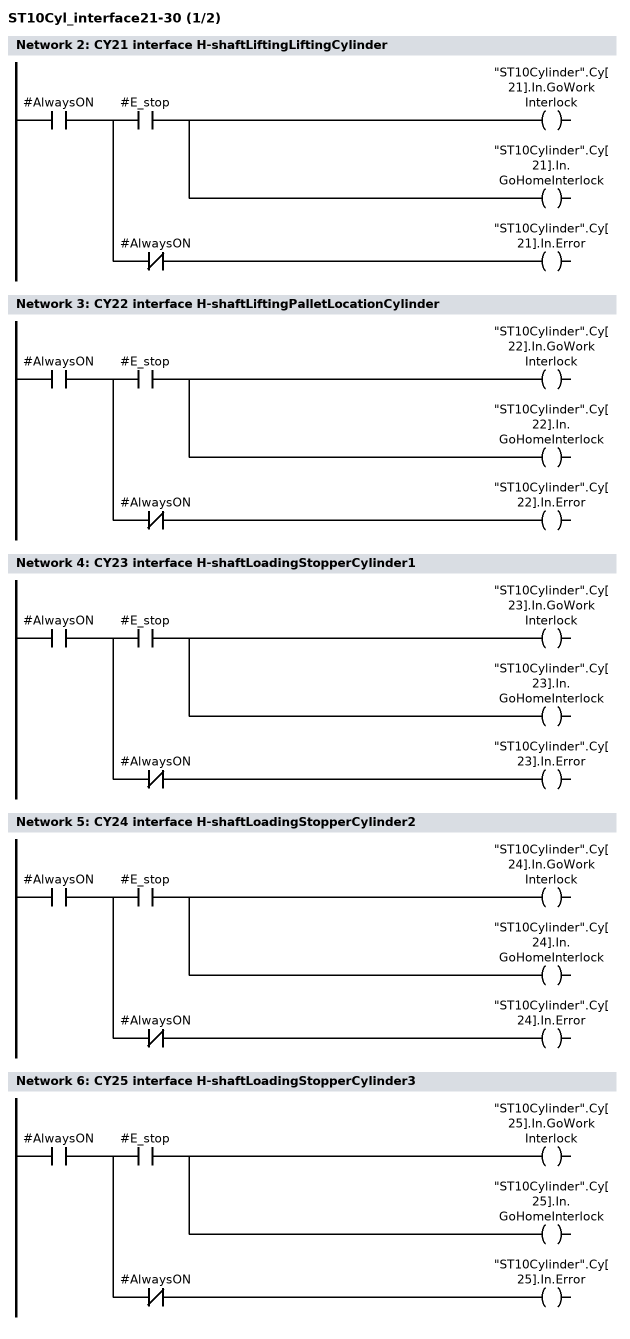
   RUNG wire#powerrail
      Contact( #AlwaysON )
      wire#w1
      Contact( #E_stop )
      wire#w2
      Coil( "ST10Cylinder".Cy[21].In.GoWorkInterlock )
   END_RUNG
   RUNG wire#w2
      Coil( "ST10Cylinder".Cy[21].In.GoHomeInterlock )
   END_RUNG
   RUNG wire#w1
      I_Contact( #AlwaysON )
      Coil( "ST10Cylinder".Cy[21].In.Error )
   END_RUNG
   // the same network as SCL:
   "ST10Cylinder".Cy[21].In.GoWorkInterlock := #AlwaysON AND #E_stop;
   "ST10Cylinder".Cy[21].In.GoHomeInterlock := #AlwaysON AND #E_stop;
   "ST10Cylinder".Cy[21].In.Error := #AlwaysON AND NOT #AlwaysON;
END_REGION

REGION Network 3: CY22 interface H-shaftLiftingPalletLocationCylinder
   RUNG wire#powerrail
      Contact( #AlwaysON )
      wire#w1
      Contact( #E_stop )
      wire#w2
      Coil( "ST10Cylinder".Cy[22].In.GoWorkInterlock )
   END_RUNG
   RUNG wire#w2
      Coil( "ST10Cylinder".Cy[22].In.GoHomeInterlock )
   END_RUNG
   RUNG wire#w1
      I_Contact( #AlwaysON )
      Coil( "ST10Cylinder".Cy[22].In.Error )
   END_RUNG
   // the same network as SCL:
   "ST10Cylinder".Cy[22].In.GoWorkInterlock := #AlwaysON AND #E_stop;
   "ST10Cylinder".Cy[22].In.GoHomeInterlock := #AlwaysON AND #E_stop;
   "ST10Cylinder".Cy[22].In.Error := #AlwaysON AND NOT #AlwaysON;
END_REGION

REGION Network 4: CY23 interface H-shaftLoadingStopperCylinder1
   RUNG wire#powerrail
      Contact( #AlwaysON )
      wire#w1
      Contact( #E_stop )
      wire#w2
      Coil( "ST10Cylinder".Cy[23].In.GoWorkInterlock )
   END_RUNG
   RUNG wire#w2
      Coil( "ST10Cylinder".Cy[23].In.GoHomeInterlock )
   END_RUNG
   RUNG wire#w1
      I_Contact( #AlwaysON )
      Coil( "ST10Cylinder".Cy[23].In.Error )
   END_RUNG
   // the same network as SCL:
   "ST10Cylinder".Cy[23].In.GoWorkInterlock := #AlwaysON AND #E_stop;
   "ST10Cylinder".Cy[23].In.GoHomeInterlock := #AlwaysON AND #E_stop;
   "ST10Cylinder".Cy[23].In.Error := #AlwaysON AND NOT #AlwaysON;
END_REGION

REGION Network 5: CY24 interface H-shaftLoadingStopperCylinder2
   RUNG wire#powerrail
      Contact( #AlwaysON )
      wire#w1
      Contact( #E_stop )
      wire#w2
      Coil( "ST10Cylinder".Cy[24].In.GoWorkInterlock )
   END_RUNG
   RUNG wire#w2
      Coil( "ST10Cylinder".Cy[24].In.GoHomeInterlock )
   END_RUNG
   RUNG wire#w1
      I_Contact( #AlwaysON )
      Coil( "ST10Cylinder".Cy[24].In.Error )
   END_RUNG
   // the same network as SCL:
   "ST10Cylinder".Cy[24].In.GoWorkInterlock := #AlwaysON AND #E_stop;
   "ST10Cylinder".Cy[24].In.GoHomeInterlock := #AlwaysON AND #E_stop;
   "ST10Cylinder".Cy[24].In.Error := #AlwaysON AND NOT #AlwaysON;
END_REGION

REGION Network 6: CY25 interface H-shaftLoadingStopperCylinder3
   RUNG wire#powerrail
      Contact( #AlwaysON )
      wire#w1
      Contact( #E_stop )
      wire#w2
      Coil( "ST10Cylinder".Cy[25].In.GoWorkInterlock )
   END_RUNG
   RUNG wire#w2
      Coil( "ST10Cylinder".Cy[25].In.GoHomeInterlock )
   END_RUNG
   RUNG wire#w1
      I_Contact( #AlwaysON )
      Coil( "ST10Cylinder".Cy[25].In.Error )
   END_RUNG
   // the same network as SCL:
   "ST10Cylinder".Cy[25].In.GoWorkInterlock := #AlwaysON AND #E_stop;
   "ST10Cylinder".Cy[25].In.GoHomeInterlock := #AlwaysON AND #E_stop;
   "ST10Cylinder".Cy[25].In.Error := #AlwaysON AND NOT #AlwaysON;
END_REGION

